LIN {X 0,Y 270.263,Z 149.626,A -85,B 0,C 180,E1 -17972.145,E2 -17972.145} C_VEL
LIN {X 0,Y 270.276,Z 149.627,A -85,B 0,C 180,E1 -17975.519,E2 -17975.519} C_VEL
LIN {X 0,Y 270.3,Z 149.622,A -85,B 0,C 180,E1 -17980.244,E2 -17980.244} C_VEL
LIN {X 0,Y 270.402,Z 149.614,A -85,B 0,C 180,E1 -17984.935,E2 -17984.935} C_VEL
LIN {X 0,Y 270.441,Z 149.602,A -85,B 0,C 180,E1 -17989.519,E2 -17989.519} C_VEL
LIN {X 0,Y 270.61,Z 149.58,A -85,B 0,C 180,E1 -17992.539,E2 -17992.539} C_VEL
LIN {X 0,Y 270.425,Z 149.61,A -85,B 0,C 180,E1 -17995.574,E2 -17995.574} C_VEL
LIN {X 0,Y 269.881,Z 149.678,A -85,B 0,C 180,E1 -17996.821,E2 -17996.821} C_VEL
LIN {X 0,Y 267.222,Z 150.002,A -85,B 0,C 180,E1 -17998.858,E2 -17998.858} C_VEL
LIN {X 0,Y 264.03,Z 150.39,A -85,B 0,C 180,E1 -18001.361,E2 -18001.361} C_VEL
LIN {X 0,Y 263.641,Z 150.441,A -85,B 0,C 180,E1 -18002.225,E2 -18002.225} C_VEL
LIN {X 0,Y 263.572,Z 150.462,A -85,B 0,C 180,E1 -18007.661,E2 -18007.661} C_VEL
LIN {X 0,Y 263.372,Z 150.472,A -85,B 0,C 180,E1 -18010.765,E2 -18010.765} C_VEL
LIN {X 0,Y 263.349,Z 150.494,A -85,B 0,C 180,E1 -18015.478,E2 -18015.478} C_VEL
LIN {X 0,Y 263.262,Z 150.491,A -85,B 0,C 180,E1 -18020.307,E2 -18020.307} C_VEL
LIN {X 0,Y 263.208,Z 150.508,A -85,B 0,C 180,E1 -18025.291,E2 -18025.291} C_VEL
LIN {X 0,Y 263.178,Z 150.505,A -85,B 0,C 180,E1 -18028.729,E2 -18028.729} C_VEL
LIN {X 0,Y 263.131,Z 150.521,A -85,B 0,C 180,E1 -18032.288,E2 -18032.288} C_VEL
LIN {X 0,Y 263.181,Z 150.514,A -85,B 0,C 180,E1 -18036.763,E2 -18036.763} C_VEL
LIN {X 0,Y 263.122,Z 150.503,A -85,B 0,C 180,E1 -18041.594,E2 -18041.594} C_VEL
LIN {X 0,Y 263.103,Z 150.515,A -85,B 0,C 180,E1 -18046.155,E2 -18046.155} C_VEL
LIN {X 0,Y 263.104,Z 150.514,A -85,B 0,C 180,E1 -18050.128,E2 -18050.128} C_VEL
LIN {X 0,Y 263.173,Z 150.515,A -85,B 0,C 180,E1 -18054.02,E2 -18054.02} C_VEL
LIN {X 0,Y 263.132,Z 150.511,A -85,B 0,C 180,E1 -18057.712,E2 -18057.712} C_VEL
LIN {X 0,Y 263.195,Z 150.632,A -85,B 0,C 180,E1 -18059.513,E2 -18059.513} C_VEL
LIN {X 0,Y 264.963,Z 158.96,A -85,B 0,C 180,E1 -18063.198,E2 -18063.198} C_VEL
LIN {X 0,Y 266.098,Z 165.732,A -85,B 0,C 180,E1 -18065.939,E2 -18065.939} C_VEL
LIN {X 0,Y 267.006,Z 169.677,A -85,B 0,C 180,E1 -18066.216,E2 -18066.216} C_VEL
LIN {X 0,Y 271.261,Z 194.933,A -85,B 0,C 180,E1 -18067.321,E2 -18067.321} C_VEL
LIN {X 0,Y 272.596,Z 205.287,A -85,B 0,C 180,E1 -18067.726,E2 -18067.726} C_VEL
LIN {X 0,Y 271.585,Z 243.518,A -85,B 0,C 180,E1 -18068.76,E2 -18068.76} C_VEL
LIN {X 0,Y 270.816,Z 255.136,A -85,B 0,C 180,E1 -18069.326,E2 -18069.326} C_VEL
LIN {X 0,Y 269.739,Z 266.296,A -85,B 0,C 180,E1 -18070.202,E2 -18070.202} C_VEL
LIN {X 0,Y 268.738,Z 274.976,A -85,B 0,C 180,E1 -18071.118,E2 -18071.118} C_VEL
LIN {X 0,Y 267.584,Z 283.269,A -85,B 0,C 180,E1 -18072.223,E2 -18072.223} C_VEL
LIN {X 0,Y 266.283,Z 291.12,A -85,B 0,C 180,E1 -18073.518,E2 -18073.518} C_VEL
LIN {X 0,Y 265.051,Z 298.464,A -85,B 0,C 180,E1 -18075.018,E2 -18075.018} C_VEL
LIN {X 0,Y 263.795,Z 305.915,A -85,B 0,C 180,E1 -18076.912,E2 -18076.912} C_VEL
LIN {X 0,Y 262.756,Z 311.756,A -85,B 0,C 180,E1 -18078.819,E2 -18078.819} C_VEL
LIN {X 0,Y 262.033,Z 316.362,A -85,B 0,C 180,E1 -18080.74,E2 -18080.74} C_VEL
LIN {X 0,Y 261.591,Z 319.357,A -85,B 0,C 180,E1 -18082.28,E2 -18082.28} C_VEL
LIN {X 0,Y 261.188,Z 322.632,A -85,B 0,C 180,E1 -18084.616,E2 -18084.616} C_VEL
LIN {X 0,Y 261.069,Z 324.672,A -85,B 0,C 180,E1 -18086.914,E2 -18086.914} C_VEL
LIN {X 0,Y 261.046,Z 325.447,A -85,B 0,C 180,E1 -18088.458,E2 -18088.458} C_VEL
LIN {X 0,Y 261.082,Z 325.74,A -85,B 0,C 180,E1 -18090,E2 -18090} C_VEL
LIN {X 0,Y 261.046,Z 325.44,A -85,B 0,C 180,E1 -18091.543,E2 -18091.543} C_VEL
LIN {X 0,Y 261.07,Z 324.65,A -85,B 0,C 180,E1 -18093.087,E2 -18093.087} C_VEL
LIN {X 0,Y 261.196,Z 322.574,A -85,B 0,C 180,E1 -18095.404,E2 -18095.404} C_VEL
LIN {X 0,Y 261.578,Z 319.298,A -85,B 0,C 180,E1 -18097.721,E2 -18097.721} C_VEL
LIN {X 0,Y 262.263,Z 314.543,A -85,B 0,C 180,E1 -18100.032,E2 -18100.032} C_VEL
LIN {X 0,Y 263.137,Z 309.397,A -85,B 0,C 180,E1 -18101.946,E2 -18101.946} C_VEL
LIN {X 0,Y 263.997,Z 304.366,A -85,B 0,C 180,E1 -18103.47,E2 -18103.47} C_VEL
LIN {X 0,Y 265.045,Z 298.308,A -85,B 0,C 180,E1 -18104.983,E2 -18104.983} C_VEL
LIN {X 0,Y 266.307,Z 290.937,A -85,B 0,C 180,E1 -18106.481,E2 -18106.481} C_VEL
LIN {X 0,Y 267.569,Z 283.043,A -85,B 0,C 180,E1 -18107.779,E2 -18107.779} C_VEL
LIN {X 0,Y 268.707,Z 274.696,A -85,B 0,C 180,E1 -18108.885,E2 -18108.885} C_VEL
LIN {X 0,Y 269.913,Z 264.253,A -85,B 0,C 180,E1 -18109.961,E2 -18109.961} C_VEL
LIN {X 0,Y 270.932,Z 252.949,A -85,B 0,C 180,E1 -18110.762,E2 -18110.762} C_VEL
LIN {X 0,Y 271.601,Z 243.673,A -85,B 0,C 180,E1 -18111.197,E2 -18111.197} C_VEL
LIN {X 0,Y 272.294,Z 214.479,A -85,B 0,C 180,E1 -18112.007,E2 -18112.007} C_VEL
LIN {X 0,Y 272.336,Z 202.812,A -85,B 0,C 180,E1 -18112.328,E2 -18112.328} C_VEL
LIN {X 0,Y 268.78,Z 179.455,A -85,B 0,C 180,E1 -18113.301,E2 -18113.301} C_VEL
LIN {X 0,Y 266.173,Z 166.332,A -85,B 0,C 180,E1 -18113.944,E2 -18113.944} C_VEL
LIN {X 0,Y 266.028,Z 165.241,A -85,B 0,C 180,E1 -18114.172,E2 -18114.172} C_VEL
LIN {X 0,Y 264.547,Z 156.793,A -85,B 0,C 180,E1 -18117.688,E2 -18117.688} C_VEL
LIN {X 0,Y 263.205,Z 150.537,A -85,B 0,C 180,E1 -18120.523,E2 -18120.523} C_VEL
LIN {X 0,Y 263.152,Z 150.51,A -85,B 0,C 180,E1 -18124.115,E2 -18124.115} C_VEL
LIN {X 0,Y 263.162,Z 150.499,A -85,B 0,C 180,E1 -18127.897,E2 -18127.897} C_VEL
LIN {X 0,Y 263.124,Z 150.524,A -85,B 0,C 180,E1 -18131.894,E2 -18131.894} C_VEL
LIN {X 0,Y 263.105,Z 150.489,A -85,B 0,C 180,E1 -18136.155,E2 -18136.155} C_VEL
LIN {X 0,Y 263.106,Z 150.522,A -85,B 0,C 180,E1 -18140.128,E2 -18140.128} C_VEL
LIN {X 0,Y 263.164,Z 150.51,A -85,B 0,C 180,E1 -18144.018,E2 -18144.018} C_VEL
LIN {X 0,Y 263.134,Z 150.521,A -85,B 0,C 180,E1 -18147.712,E2 -18147.712} C_VEL
LIN {X 0,Y 263.203,Z 150.498,A -85,B 0,C 180,E1 -18151.783,E2 -18151.783} C_VEL
LIN {X 0,Y 263.228,Z 150.51,A -85,B 0,C 180,E1 -18155.2,E2 -18155.2} C_VEL
LIN {X 0,Y 263.265,Z 150.49,A -85,B 0,C 180,E1 -18159.694,E2 -18159.694} C_VEL
LIN {X 0,Y 263.353,Z 150.494,A -85,B 0,C 180,E1 -18164.522,E2 -18164.522} C_VEL
LIN {X 0,Y 263.357,Z 150.474,A -85,B 0,C 180,E1 -18169.234,E2 -18169.234} C_VEL
LIN {X 0,Y 263.56,Z 150.463,A -85,B 0,C 180,E1 -18172.338,E2 -18172.338} C_VEL
LIN {X 0,Y 263.752,Z 150.426,A -85,B 0,C 180,E1 -18178.473,E2 -18178.473} C_VEL
LIN {X 0,Y 263.753,Z 150.435,A -85,B 0,C 180,E1 -18181.527,E2 -18181.527} C_VEL
LIN {X 0,Y 263.575,Z 150.453,A -85,B 0,C 180,E1 -18187.662,E2 -18187.662} C_VEL
LIN {X 0,Y 263.377,Z 150.481,A -85,B 0,C 180,E1 -18190.766,E2 -18190.766} C_VEL
LIN {X 0,Y 263.353,Z 150.49,A -85,B 0,C 180,E1 -18195.478,E2 -18195.478} C_VEL
LIN {X 0,Y 263.266,Z 150.497,A -85,B 0,C 180,E1 -18200.307,E2 -18200.307} C_VEL
LIN {X 0,Y 263.21,Z 150.501,A -85,B 0,C 180,E1 -18205.291,E2 -18205.291} C_VEL
LIN {X 0,Y 263.181,Z 150.51,A -85,B 0,C 180,E1 -18208.73,E2 -18208.73} C_VEL
LIN {X 0,Y 263.135,Z 150.518,A -85,B 0,C 180,E1 -18212.288,E2 -18212.288} C_VEL
LIN {X 0,Y 263.185,Z 150.516,A -85,B 0,C 180,E1 -18216.763,E2 -18216.763} C_VEL
LIN {X 0,Y 263.126,Z 150.519,A -85,B 0,C 180,E1 -18221.593,E2 -18221.593} C_VEL
LIN {X 0,Y 263.124,Z 150.522,A -85,B 0,C 180,E1 -18223.984,E2 -18223.984} C_VEL
LIN {X 0,Y 263.126,Z 150.497,A -85,B 0,C 180,E1 -18228.406,E2 -18228.406} C_VEL
LIN {X 0,Y 263.167,Z 150.517,A -85,B 0,C 180,E1 -18232.104,E2 -18232.104} C_VEL
LIN {X 0,Y 263.169,Z 150.498,A -85,B 0,C 180,E1 -18235.888,E2 -18235.888} C_VEL
LIN {X 0,Y 263.153,Z 150.511,A -85,B 0,C 180,E1 -18239.507,E2 -18239.507} C_VEL
LIN {X 0,Y 263.297,Z 150.677,A -85,B 0,C 180,E1 -18243.014,E2 -18243.014} C_VEL
LIN {X 0,Y 264.578,Z 157.239,A -85,B 0,C 180,E1 -18245.894,E2 -18245.894} C_VEL
LIN {X 0,Y 266.07,Z 161.339,A -85,B 0,C 180,E1 -18246.226,E2 -18246.226} C_VEL
LIN {X 0,Y 269.712,Z 171.853,A -85,B 0,C 180,E1 -18246.868,E2 -18246.868} C_VEL
LIN {X 0,Y 272.813,Z 188.856,A -85,B 0,C 180,E1 -18247.623,E2 -18247.623} C_VEL
LIN {X 0,Y 271.762,Z 233.501,A -85,B 0,C 180,E1 -18248.823,E2 -18248.823} C_VEL
LIN {X 0,Y 271.245,Z 243.265,A -85,B 0,C 180,E1 -18249.278,E2 -18249.278} C_VEL
LIN {X 0,Y 270.43,Z 254.338,A -85,B 0,C 180,E1 -18250.056,E2 -18250.056} C_VEL
LIN {X 0,Y 269.192,Z 265.146,A -85,B 0,C 180,E1 -18251.15,E2 -18251.15} C_VEL
LIN {X 0,Y 268.087,Z 273.533,A -85,B 0,C 180,E1 -18252.256,E2 -18252.256} C_VEL
LIN {X 0,Y 266.877,Z 281.453,A -85,B 0,C 180,E1 -18253.555,E2 -18253.555} C_VEL
LIN {X 0,Y 265.981,Z 287.139,A -85,B 0,C 180,E1 -18254.679,E2 -18254.679} C_VEL
LIN {X 0,Y 264.849,Z 293.489,A -85,B 0,C 180,E1 -18256.183,E2 -18256.183} C_VEL
LIN {X 0,Y 263.923,Z 298.766,A -85,B 0,C 180,E1 -18257.7,E2 -18257.7} C_VEL
LIN {X 0,Y 263.077,Z 303.172,A -85,B 0,C 180,E1 -18259.222,E2 -18259.222} C_VEL
LIN {X 0,Y 262.253,Z 308.35,A -85,B 0,C 180,E1 -18261.524,E2 -18261.524} C_VEL
LIN {X 0,Y 261.681,Z 311.772,A -85,B 0,C 180,E1 -18263.574,E2 -18263.574} C_VEL
LIN {X 0,Y 261.381,Z 313.917,A -85,B 0,C 180,E1 -18265.373,E2 -18265.373} C_VEL
LIN {X 0,Y 261.213,Z 315.186,A -85,B 0,C 180,E1 -18266.915,E2 -18266.915} C_VEL
LIN {X 0,Y 261.099,Z 315.987,A -85,B 0,C 180,E1 -18268.457,E2 -18268.457} C_VEL
LIN {X 0,Y 261.088,Z 316.292,A -85,B 0,C 180,E1 -18270,E2 -18270} C_VEL
LIN {X 0,Y 261.099,Z 316.013,A -85,B 0,C 180,E1 -18271.542,E2 -18271.542} C_VEL
LIN {X 0,Y 261.211,Z 315.265,A -85,B 0,C 180,E1 -18273.084,E2 -18273.084} C_VEL
LIN {X 0,Y 261.371,Z 314.049,A -85,B 0,C 180,E1 -18274.627,E2 -18274.627} C_VEL
LIN {X 0,Y 261.755,Z 311.196,A -85,B 0,C 180,E1 -18276.938,E2 -18276.938} C_VEL
LIN {X 0,Y 262.2,Z 308.596,A -85,B 0,C 180,E1 -18278.477,E2 -18278.477} C_VEL
LIN {X 0,Y 263.061,Z 303.484,A -85,B 0,C 180,E1 -18280.778,E2 -18280.778} C_VEL
LIN {X 0,Y 264.072,Z 297.981,A -85,B 0,C 180,E1 -18282.683,E2 -18282.683} C_VEL
LIN {X 0,Y 265.345,Z 291.064,A -85,B 0,C 180,E1 -18284.573,E2 -18284.573} C_VEL
LIN {X 0,Y 266.64,Z 283.123,A -85,B 0,C 180,E1 -18286.263,E2 -18286.263} C_VEL
LIN {X 0,Y 267.825,Z 275.549,A -85,B 0,C 180,E1 -18287.564,E2 -18287.564} C_VEL
LIN {X 0,Y 268.995,Z 267.606,A -85,B 0,C 180,E1 -18288.666,E2 -18288.666} C_VEL
LIN {X 0,Y 269.999,Z 259.4,A -85,B 0,C 180,E1 -18289.58,E2 -18289.58} C_VEL
LIN {X 0,Y 270.786,Z 251.226,A -85,B 0,C 180,E1 -18290.3,E2 -18290.3} C_VEL
LIN {X 0,Y 271.431,Z 242.496,A -85,B 0,C 180,E1 -18290.88,E2 -18290.88} C_VEL
LIN {X 0,Y 271.86,Z 234.107,A -85,B 0,C 180,E1 -18291.272,E2 -18291.272} C_VEL
LIN {X 0,Y 272.318,Z 212.774,A -85,B 0,C 180,E1 -18291.88,E2 -18291.88} C_VEL
LIN {X 0,Y 272.859,Z 188.975,A -85,B 0,C 180,E1 -18292.497,E2 -18292.497} C_VEL
LIN {X 0,Y 269.51,Z 171.11,A -85,B 0,C 180,E1 -18293.301,E2 -18293.301} C_VEL
LIN {X 0,Y 265.613,Z 160.117,A -85,B 0,C 180,E1 -18293.984,E2 -18293.984} C_VEL
LIN {X 0,Y 264.555,Z 157.188,A -85,B 0,C 180,E1 -18294.249,E2 -18294.249} C_VEL
LIN {X 0,Y 263.312,Z 150.747,A -85,B 0,C 180,E1 -18297.078,E2 -18297.078} C_VEL
LIN {X 0,Y 263.18,Z 150.515,A -85,B 0,C 180,E1 -18298.729,E2 -18298.729} C_VEL
LIN {X 0,Y 263.134,Z 150.522,A -85,B 0,C 180,E1 -18302.288,E2 -18302.288} C_VEL
LIN {X 0,Y 263.187,Z 150.497,A -85,B 0,C 180,E1 -18305.977,E2 -18305.977} C_VEL
LIN {X 0,Y 263.115,Z 150.517,A -85,B 0,C 180,E1 -18309.87,E2 -18309.87} C_VEL
LIN {X 0,Y 263.103,Z 150.504,A -85,B 0,C 180,E1 -18313.988,E2 -18313.988} C_VEL
LIN {X 0,Y 263.123,Z 150.521,A -85,B 0,C 180,E1 -18318.106,E2 -18318.106} C_VEL
LIN {X 0,Y 263.158,Z 150.516,A -85,B 0,C 180,E1 -18322.103,E2 -18322.103} C_VEL
LIN {X 0,Y 263.15,Z 150.507,A -85,B 0,C 180,E1 -18325.885,E2 -18325.885} C_VEL
LIN {X 0,Y 263.15,Z 150.519,A -85,B 0,C 180,E1 -18329.507,E2 -18329.507} C_VEL
LIN {X 0,Y 263.191,Z 150.502,A -85,B 0,C 180,E1 -18333.002,E2 -18333.002} C_VEL
LIN {X 0,Y 263.183,Z 150.511,A -85,B 0,C 180,E1 -18336.387,E2 -18336.387} C_VEL
LIN {X 0,Y 263.263,Z 150.498,A -85,B 0,C 180,E1 -18339.693,E2 -18339.693} C_VEL
LIN {X 0,Y 263.35,Z 150.49,A -85,B 0,C 180,E1 -18344.522,E2 -18344.522} C_VEL
LIN {X 0,Y 263.373,Z 150.481,A -85,B 0,C 180,E1 -18349.234,E2 -18349.234} C_VEL
LIN {X 0,Y 263.571,Z 150.453,A -85,B 0,C 180,E1 -18352.338,E2 -18352.338} C_VEL
LIN {X 0,Y 263.751,Z 150.436,A -85,B 0,C 180,E1 -18358.473,E2 -18358.473} C_VEL
LIN {X 0,Y 263.75,Z 150.426,A -85,B 0,C 180,E1 -18361.527,E2 -18361.527} C_VEL
LIN {X 0,Y 263.641,Z 150.441,A -85,B 0,C 180,E1 -18362.225,E2 -18362.225} C_VEL
LIN {X 0,Y 262.865,Z 150.549,A -85,B 0,C 180,E1 -18363.499,E2 -18363.499} C_VEL
LIN {X 0,Y 259.97,Z 150.915,A -85,B 0,C 180,E1 -18365.576,E2 -18365.576} C_VEL
LIN {X 0,Y 257.579,Z 151.211,A -85,B 0,C 180,E1 -18367.264,E2 -18367.264} C_VEL
LIN {X 0,Y 256.559,Z 151.33,A -85,B 0,C 180,E1 -18368.574,E2 -18368.574} C_VEL
LIN {X 0,Y 256.476,Z 151.335,A -85,B 0,C 180,E1 -18369.017,E2 -18369.017} C_VEL
LIN {X 0,Y 256.294,Z 151.365,A -85,B 0,C 180,E1 -18372.672,E2 -18372.672} C_VEL
LIN {X 0,Y 256.281,Z 151.371,A -85,B 0,C 180,E1 -18376.302,E2 -18376.302} C_VEL
LIN {X 0,Y 256.156,Z 151.38,A -85,B 0,C 180,E1 -18381.12,E2 -18381.12} C_VEL
LIN {X 0,Y 256.187,Z 151.383,A -85,B 0,C 180,E1 -18385.139,E2 -18385.139} C_VEL
LIN {X 0,Y 256.112,Z 151.392,A -85,B 0,C 180,E1 -18389.6,E2 -18389.6} C_VEL
LIN {X 0,Y 256.066,Z 151.395,A -85,B 0,C 180,E1 -18393.293,E2 -18393.293} C_VEL
LIN {X 0,Y 256.113,Z 151.395,A -85,B 0,C 180,E1 -18397.271,E2 -18397.271} C_VEL
LIN {X 0,Y 256.052,Z 151.387,A -85,B 0,C 180,E1 -18401.204,E2 -18401.204} C_VEL
LIN {X 0,Y 256.039,Z 151.391,A -85,B 0,C 180,E1 -18405.534,E2 -18405.534} C_VEL
LIN {X 0,Y 256.053,Z 151.4,A -85,B 0,C 180,E1 -18408.797,E2 -18408.797} C_VEL
LIN {X 0,Y 256.134,Z 151.379,A -85,B 0,C 180,E1 -18412.869,E2 -18412.869} C_VEL
LIN {X 0,Y 256.067,Z 151.388,A -85,B 0,C 180,E1 -18416.708,E2 -18416.708} C_VEL
LIN {X 0,Y 256.126,Z 151.528,A -85,B 0,C 180,E1 -18419.037,E2 -18419.037} C_VEL
LIN {X 0,Y 257.709,Z 158.819,A -85,B 0,C 180,E1 -18422.38,E2 -18422.38} C_VEL
LIN {X 0,Y 258.959,Z 165.635,A -85,B 0,C 180,E1 -18425.239,E2 -18425.239} C_VEL
LIN {X 0,Y 260.509,Z 170.647,A -85,B 0,C 180,E1 -18425.616,E2 -18425.616} C_VEL
LIN {X 0,Y 265.165,Z 198.563,A -85,B 0,C 180,E1 -18426.877,E2 -18426.877} C_VEL
LIN {X 0,Y 266.018,Z 205.812,A -85,B 0,C 180,E1 -18427.163,E2 -18427.163} C_VEL
LIN {X 0,Y 265.042,Z 242.239,A -85,B 0,C 180,E1 -18428.163,E2 -18428.163} C_VEL
LIN {X 0,Y 264.452,Z 251.768,A -85,B 0,C 180,E1 -18428.602,E2 -18428.602} C_VEL
LIN {X 0,Y 263.459,Z 262.934,A -85,B 0,C 180,E1 -18429.38,E2 -18429.38} C_VEL
LIN {X 0,Y 262.208,Z 273.349,A -85,B 0,C 180,E1 -18430.426,E2 -18430.426} C_VEL
LIN {X 0,Y 261.025,Z 281.914,A -85,B 0,C 180,E1 -18431.557,E2 -18431.557} C_VEL
LIN {X 0,Y 259.635,Z 289.972,A -85,B 0,C 180,E1 -18432.881,E2 -18432.881} C_VEL
LIN {X 0,Y 258.496,Z 296.631,A -85,B 0,C 180,E1 -18434.224,E2 -18434.224} C_VEL
LIN {X 0,Y 257.33,Z 302.953,A -85,B 0,C 180,E1 -18435.771,E2 -18435.771} C_VEL
LIN {X 0,Y 256.389,Z 308.207,A -85,B 0,C 180,E1 -18437.333,E2 -18437.333} C_VEL
LIN {X 0,Y 255.609,Z 312.588,A -85,B 0,C 180,E1 -18438.904,E2 -18438.904} C_VEL
LIN {X 0,Y 254.777,Z 317.758,A -85,B 0,C 180,E1 -18441.274,E2 -18441.274} C_VEL
LIN {X 0,Y 254.207,Z 321.552,A -85,B 0,C 180,E1 -18443.651,E2 -18443.651} C_VEL
LIN {X 0,Y 254.061,Z 323.296,A -85,B 0,C 180,E1 -18445.24,E2 -18445.24} C_VEL
LIN {X 0,Y 253.972,Z 324.544,A -85,B 0,C 180,E1 -18446.828,E2 -18446.828} C_VEL
LIN {X 0,Y 253.957,Z 325.319,A -85,B 0,C 180,E1 -18448.415,E2 -18448.415} C_VEL
LIN {X 0,Y 253.989,Z 325.612,A -85,B 0,C 180,E1 -18450,E2 -18450} C_VEL
LIN {X 0,Y 253.957,Z 325.311,A -85,B 0,C 180,E1 -18451.586,E2 -18451.586} C_VEL
LIN {X 0,Y 253.972,Z 324.521,A -85,B 0,C 180,E1 -18453.173,E2 -18453.173} C_VEL
LIN {X 0,Y 254.085,Z 322.726,A -85,B 0,C 180,E1 -18455.279,E2 -18455.279} C_VEL
LIN {X 0,Y 254.544,Z 319.168,A -85,B 0,C 180,E1 -18457.935,E2 -18457.935} C_VEL
LIN {X 0,Y 255.256,Z 314.413,A -85,B 0,C 180,E1 -18460.31,E2 -18460.31} C_VEL
LIN {X 0,Y 256.171,Z 309.266,A -85,B 0,C 180,E1 -18462.276,E2 -18462.276} C_VEL
LIN {X 0,Y 257.076,Z 304.235,A -85,B 0,C 180,E1 -18463.84,E2 -18463.84} C_VEL
LIN {X 0,Y 258.169,Z 298.177,A -85,B 0,C 180,E1 -18465.392,E2 -18465.392} C_VEL
LIN {X 0,Y 259.502,Z 290.806,A -85,B 0,C 180,E1 -18466.926,E2 -18466.926} C_VEL
LIN {X 0,Y 260.825,Z 282.911,A -85,B 0,C 180,E1 -18468.255,E2 -18468.255} C_VEL
LIN {X 0,Y 261.998,Z 274.563,A -85,B 0,C 180,E1 -18469.388,E2 -18469.388} C_VEL
LIN {X 0,Y 263.233,Z 264.33,A -85,B 0,C 180,E1 -18470.469,E2 -18470.469} C_VEL
LIN {X 0,Y 264.313,Z 252.944,A -85,B 0,C 180,E1 -18471.299,E2 -18471.299} C_VEL
LIN {X 0,Y 265,Z 243.247,A -85,B 0,C 180,E1 -18471.762,E2 -18471.762} C_VEL
LIN {X 0,Y 265.875,Z 204.461,A -85,B 0,C 180,E1 -18472.85,E2 -18472.85} C_VEL
LIN {X 0,Y 262.258,Z 180.54,A -85,B 0,C 180,E1 -18473.88,E2 -18473.88} C_VEL
LIN {X 0,Y 259.863,Z 168.483,A -85,B 0,C 180,E1 -18474.47,E2 -18474.47} C_VEL
LIN {X 0,Y 258.933,Z 165.659,A -85,B 0,C 180,E1 -18474.718,E2 -18474.718} C_VEL
LIN {X 0,Y 257.699,Z 158.712,A -85,B 0,C 180,E1 -18477.622,E2 -18477.622} C_VEL
LIN {X 0,Y 256.14,Z 151.436,A -85,B 0,C 180,E1 -18480.991,E2 -18480.991} C_VEL
LIN {X 0,Y 256.089,Z 151.398,A -85,B 0,C 180,E1 -18485.192,E2 -18485.192} C_VEL
LIN {X 0,Y 256.121,Z 151.379,A -85,B 0,C 180,E1 -18487.273,E2 -18487.273} C_VEL
LIN {X 0,Y 256.055,Z 151.4,A -85,B 0,C 180,E1 -18491.204,E2 -18491.204} C_VEL
LIN {X 0,Y 256.041,Z 151.371,A -85,B 0,C 180,E1 -18495.534,E2 -18495.534} C_VEL
LIN {X 0,Y 256.055,Z 151.388,A -85,B 0,C 180,E1 -18498.797,E2 -18498.797} C_VEL
LIN {X 0,Y 256.132,Z 151.392,A -85,B 0,C 180,E1 -18502.868,E2 -18502.868} C_VEL
LIN {X 0,Y 256.069,Z 151.395,A -85,B 0,C 180,E1 -18506.708,E2 -18506.708} C_VEL
LIN {X 0,Y 256.115,Z 151.391,A -85,B 0,C 180,E1 -18510.401,E2 -18510.401} C_VEL
LIN {X 0,Y 256.19,Z 151.383,A -85,B 0,C 180,E1 -18514.861,E2 -18514.861} C_VEL
LIN {X 0,Y 256.168,Z 151.376,A -85,B 0,C 180,E1 -18519.105,E2 -18519.105} C_VEL
LIN {X 0,Y 256.302,Z 151.37,A -85,B 0,C 180,E1 -18524.085,E2 -18524.085} C_VEL
LIN {X 0,Y 256.299,Z 151.353,A -85,B 0,C 180,E1 -18528.934,E2 -18528.934} C_VEL
LIN {X 0,Y 256.517,Z 151.338,A -85,B 0,C 180,E1 -18532.127,E2 -18532.127} C_VEL
LIN {X 0,Y 256.499,Z 151.339,A -85,B 0,C 180,E1 -18536.859,E2 -18536.859} C_VEL
LIN {X 0,Y 256.76,Z 151.296,A -85,B 0,C 180,E1 -18540,E2 -18540} C_VEL
LIN {X 0,Y 256.5,Z 151.344,A -85,B 0,C 180,E1 -18543.142,E2 -18543.142} C_VEL
LIN {X 0,Y 256.542,Z 151.326,A -85,B 0,C 180,E1 -18547.873,E2 -18547.873} C_VEL
LIN {X 0,Y 256.313,Z 151.361,A -85,B 0,C 180,E1 -18551.066,E2 -18551.066} C_VEL
LIN {X 0,Y 256.302,Z 151.365,A -85,B 0,C 180,E1 -18555.915,E2 -18555.915} C_VEL
LIN {X 0,Y 256.169,Z 151.383,A -85,B 0,C 180,E1 -18560.895,E2 -18560.895} C_VEL
LIN {X 0,Y 256.19,Z 151.376,A -85,B 0,C 180,E1 -18565.138,E2 -18565.138} C_VEL
LIN {X 0,Y 256.116,Z 151.394,A -85,B 0,C 180,E1 -18569.6,E2 -18569.6} C_VEL
LIN {X 0,Y 256.07,Z 151.388,A -85,B 0,C 180,E1 -18573.293,E2 -18573.293} C_VEL
LIN {X 0,Y 256.117,Z 151.394,A -85,B 0,C 180,E1 -18577.271,E2 -18577.271} C_VEL
LIN {X 0,Y 256.056,Z 151.4,A -85,B 0,C 180,E1 -18581.203,E2 -18581.203} C_VEL
LIN {X 0,Y 256.046,Z 151.391,A -85,B 0,C 180,E1 -18585.533,E2 -18585.533} C_VEL
LIN {X 0,Y 256.058,Z 151.379,A -85,B 0,C 180,E1 -18588.797,E2 -18588.797} C_VEL
LIN {X 0,Y 256.146,Z 151.387,A -85,B 0,C 180,E1 -18592.87,E2 -18592.87} C_VEL
LIN {X 0,Y 256.078,Z 151.39,A -85,B 0,C 180,E1 -18596.708,E2 -18596.708} C_VEL
LIN {X 0,Y 256.141,Z 151.392,A -85,B 0,C 180,E1 -18601.404,E2 -18601.404} C_VEL
LIN {X 0,Y 256.265,Z 151.551,A -85,B 0,C 180,E1 -18602.543,E2 -18602.543} C_VEL
LIN {X 0,Y 257.41,Z 157.377,A -85,B 0,C 180,E1 -18605.177,E2 -18605.177} C_VEL
LIN {X 0,Y 258.898,Z 161.415,A -85,B 0,C 180,E1 -18605.522,E2 -18605.522} C_VEL
LIN {X 0,Y 263.102,Z 172.815,A -85,B 0,C 180,E1 -18606.275,E2 -18606.275} C_VEL
LIN {X 0,Y 266.181,Z 189.334,A -85,B 0,C 180,E1 -18607.043,E2 -18607.043} C_VEL
LIN {X 0,Y 265.392,Z 227.395,A -85,B 0,C 180,E1 -18608.064,E2 -18608.064} C_VEL
LIN {X 0,Y 264.843,Z 240.179,A -85,B 0,C 180,E1 -18608.555,E2 -18608.555} C_VEL
LIN {X 0,Y 264.174,Z 249.7,A -85,B 0,C 180,E1 -18609.159,E2 -18609.159} C_VEL
LIN {X 0,Y 263.367,Z 258.335,A -85,B 0,C 180,E1 -18609.905,E2 -18609.905} C_VEL
LIN {X 0,Y 262.298,Z 266.777,A -85,B 0,C 180,E1 -18610.839,E2 -18610.839} C_VEL
LIN {X 0,Y 261.148,Z 274.894,A -85,B 0,C 180,E1 -18611.971,E2 -18611.971} C_VEL
LIN {X 0,Y 259.941,Z 282.604,A -85,B 0,C 180,E1 -18613.305,E2 -18613.305} C_VEL
LIN {X 0,Y 258.556,Z 290.666,A -85,B 0,C 180,E1 -18615.035,E2 -18615.035} C_VEL
LIN {X 0,Y 257.193,Z 297.727,A -85,B 0,C 180,E1 -18616.971,E2 -18616.971} C_VEL
LIN {X 0,Y 256.09,Z 303.303,A -85,B 0,C 180,E1 -18618.924,E2 -18618.924} C_VEL
LIN {X 0,Y 255.227,Z 308.48,A -85,B 0,C 180,E1 -18621.289,E2 -18621.289} C_VEL
LIN {X 0,Y 254.605,Z 312.168,A -85,B 0,C 180,E1 -18623.58,E2 -18623.58} C_VEL
LIN {X 0,Y 254.304,Z 314.046,A -85,B 0,C 180,E1 -18625.244,E2 -18625.244} C_VEL
LIN {X 0,Y 254.135,Z 315.315,A -85,B 0,C 180,E1 -18626.829,E2 -18626.829} C_VEL
LIN {X 0,Y 254.011,Z 316.116,A -85,B 0,C 180,E1 -18628.414,E2 -18628.414} C_VEL
LIN {X 0,Y 254.018,Z 316.42,A -85,B 0,C 180,E1 -18630,E2 -18630} C_VEL
LIN {X 0,Y 254.011,Z 316.141,A -85,B 0,C 180,E1 -18631.585,E2 -18631.585} C_VEL
LIN {X 0,Y 254.132,Z 315.393,A -85,B 0,C 180,E1 -18633.17,E2 -18633.17} C_VEL
LIN {X 0,Y 254.291,Z 314.176,A -85,B 0,C 180,E1 -18634.756,E2 -18634.756} C_VEL
LIN {X 0,Y 254.53,Z 312.47,A -85,B 0,C 180,E1 -18636.341,E2 -18636.341} C_VEL
LIN {X 0,Y 255.189,Z 308.723,A -85,B 0,C 180,E1 -18638.712,E2 -18638.712} C_VEL
LIN {X 0,Y 256.078,Z 303.611,A -85,B 0,C 180,E1 -18641.076,E2 -18641.076} C_VEL
LIN {X 0,Y 257.139,Z 298.107,A -85,B 0,C 180,E1 -18643.031,E2 -18643.031} C_VEL
LIN {X 0,Y 258.496,Z 291.19,A -85,B 0,C 180,E1 -18644.968,E2 -18644.968} C_VEL
LIN {X 0,Y 259.833,Z 283.248,A -85,B 0,C 180,E1 -18646.701,E2 -18646.701} C_VEL
LIN {X 0,Y 261.087,Z 275.673,A -85,B 0,C 180,E1 -18648.032,E2 -18648.032} C_VEL
LIN {X 0,Y 262.296,Z 267.729,A -85,B 0,C 180,E1 -18649.161,E2 -18649.161} C_VEL
LIN {X 0,Y 263.343,Z 259.522,A -85,B 0,C 180,E1 -18650.096,E2 -18650.096} C_VEL
LIN {X 0,Y 264.235,Z 250.538,A -85,B 0,C 180,E1 -18650.894,E2 -18650.894} C_VEL
LIN {X 0,Y 264.914,Z 241.079,A -85,B 0,C 180,E1 -18651.513,E2 -18651.513} C_VEL
LIN {X 0,Y 265.318,Z 230.589,A -85,B 0,C 180,E1 -18651.966,E2 -18651.966} C_VEL
LIN {X 0,Y 266.315,Z 189.944,A -85,B 0,C 180,E1 -18653.056,E2 -18653.056} C_VEL
LIN {X 0,Y 263.257,Z 173.419,A -85,B 0,C 180,E1 -18653.823,E2 -18653.823} C_VEL
LIN {X 0,Y 259.585,Z 163.09,A -85,B 0,C 180,E1 -18654.491,E2 -18654.491} C_VEL
LIN {X 0,Y 257.467,Z 157.603,A -85,B 0,C 180,E1 -18654.916,E2 -18654.916} C_VEL
LIN {X 0,Y 257.227,Z 156.464,A -85,B 0,C 180,E1 -18655.272,E2 -18655.272} C_VEL
LIN {X 0,Y 256.213,Z 151.476,A -85,B 0,C 180,E1 -18657.684,E2 -18657.684} C_VEL
LIN {X 0,Y 256.084,Z 151.398,A -85,B 0,C 180,E1 -18661.704,E2 -18661.704} C_VEL
LIN {X 0,Y 256.12,Z 151.372,A -85,B 0,C 180,E1 -18665.186,E2 -18665.186} C_VEL
LIN {X 0,Y 256.088,Z 151.397,A -85,B 0,C 180,E1 -18669.138,E2 -18669.138} C_VEL
LIN {X 0,Y 256.048,Z 151.373,A -85,B 0,C 180,E1 -18673.329,E2 -18673.329} C_VEL
LIN {X 0,Y 256.071,Z 151.401,A -85,B 0,C 180,E1 -18677.818,E2 -18677.818} C_VEL
LIN {X 0,Y 256.07,Z 151.392,A -85,B 0,C 180,E1 -18680.858,E2 -18680.858} C_VEL
LIN {X 0,Y 256.13,Z 151.393,A -85,B 0,C 180,E1 -18682.867,E2 -18682.867} C_VEL
LIN {X 0,Y 256.067,Z 151.388,A -85,B 0,C 180,E1 -18686.707,E2 -18686.707} C_VEL
LIN {X 0,Y 256.113,Z 151.394,A -85,B 0,C 180,E1 -18690.4,E2 -18690.4} C_VEL
LIN {X 0,Y 256.187,Z 151.376,A -85,B 0,C 180,E1 -18694.861,E2 -18694.861} C_VEL
LIN {X 0,Y 256.166,Z 151.384,A -85,B 0,C 180,E1 -18699.105,E2 -18699.105} C_VEL
LIN {X 0,Y 256.299,Z 151.364,A -85,B 0,C 180,E1 -18704.085,E2 -18704.085} C_VEL
LIN {X 0,Y 256.309,Z 151.362,A -85,B 0,C 180,E1 -18708.934,E2 -18708.934} C_VEL
LIN {X 0,Y 256.539,Z 151.326,A -85,B 0,C 180,E1 -18712.127,E2 -18712.127} C_VEL
LIN {X 0,Y 256.713,Z 151.312,A -85,B 0,C 180,E1 -18718.431,E2 -18718.431} C_VEL
LIN {X 0,Y 256.713,Z 151.301,A -85,B 0,C 180,E1 -18721.569,E2 -18721.569} C_VEL
LIN {X 0,Y 256.539,Z 151.336,A -85,B 0,C 180,E1 -18727.873,E2 -18727.873} C_VEL
LIN {X 0,Y 256.476,Z 151.335,A -85,B 0,C 180,E1 -18729.017,E2 -18729.017} C_VEL
LIN {X 0,Y 255.772,Z 151.423,A -85,B 0,C 180,E1 -18730.326,E2 -18730.326} C_VEL
LIN {X 0,Y 252.797,Z 151.8,A -85,B 0,C 180,E1 -18732.455,E2 -18732.455} C_VEL
LIN {X 0,Y 250.303,Z 152.117,A -85,B 0,C 180,E1 -18734.189,E2 -18734.189} C_VEL
LIN {X 0,Y 249.275,Z 152.247,A -85,B 0,C 180,E1 -18735.537,E2 -18735.537} C_VEL
LIN {X 0,Y 249.213,Z 152.25,A -85,B 0,C 180,E1 -18735.994,E2 -18735.994} C_VEL
LIN {X 0,Y 249.109,Z 152.251,A -85,B 0,C 180,E1 -18739.788,E2 -18739.788} C_VEL
LIN {X 0,Y 249.15,Z 152.26,A -85,B 0,C 180,E1 -18745.031,E2 -18745.031} C_VEL
LIN {X 0,Y 249.082,Z 152.262,A -85,B 0,C 180,E1 -18748.994,E2 -18748.994} C_VEL
LIN {X 0,Y 249.029,Z 152.278,A -85,B 0,C 180,E1 -18752.426,E2 -18752.426} C_VEL
LIN {X 0,Y 249.046,Z 152.27,A -85,B 0,C 180,E1 -18756.342,E2 -18756.342} C_VEL
LIN {X 0,Y 249.004,Z 152.268,A -85,B 0,C 180,E1 -18760.478,E2 -18760.478} C_VEL
LIN {X 0,Y 248.983,Z 152.255,A -85,B 0,C 180,E1 -18764.883,E2 -18764.883} C_VEL
LIN {X 0,Y 249.008,Z 152.278,A -85,B 0,C 180,E1 -18767.362,E2 -18767.362} C_VEL
LIN {X 0,Y 249.026,Z 152.257,A -85,B 0,C 180,E1 -18771.62,E2 -18771.62} C_VEL
LIN {X 0,Y 249.044,Z 152.269,A -85,B 0,C 180,E1 -18775.64,E2 -18775.64} C_VEL
LIN {X 0,Y 249.07,Z 152.424,A -85,B 0,C 180,E1 -18778.533,E2 -18778.533} C_VEL
LIN {X 0,Y 250.685,Z 159.727,A -85,B 0,C 180,E1 -18781.993,E2 -18781.993} C_VEL
LIN {X 0,Y 251.78,Z 165.508,A -85,B 0,C 180,E1 -18784.485,E2 -18784.485} C_VEL
LIN {X 0,Y 253.816,Z 171.355,A -85,B 0,C 180,E1 -18784.955,E2 -18784.955} C_VEL
LIN {X 0,Y 256.597,Z 186.358,A -85,B 0,C 180,E1 -18785.695,E2 -18785.695} C_VEL
LIN {X 0,Y 259.485,Z 206.407,A -85,B 0,C 180,E1 -18786.575,E2 -18786.575} C_VEL
LIN {X 0,Y 258.484,Z 241.852,A -85,B 0,C 180,E1 -18787.568,E2 -18787.568} C_VEL
LIN {X 0,Y 257.882,Z 251.094,A -85,B 0,C 180,E1 -18787.994,E2 -18787.994} C_VEL
LIN {X 0,Y 257.073,Z 260.281,A -85,B 0,C 180,E1 -18788.623,E2 -18788.623} C_VEL
LIN {X 0,Y 255.96,Z 269.798,A -85,B 0,C 180,E1 -18789.508,E2 -18789.508} C_VEL
LIN {X 0,Y 254.481,Z 280.557,A -85,B 0,C 180,E1 -18790.856,E2 -18790.856} C_VEL
LIN {X 0,Y 253.078,Z 288.825,A -85,B 0,C 180,E1 -18792.214,E2 -18792.214} C_VEL
LIN {X 0,Y 251.666,Z 296.505,A -85,B 0,C 180,E1 -18793.784,E2 -18793.784} C_VEL
LIN {X 0,Y 250.432,Z 302.826,A -85,B 0,C 180,E1 -18795.371,E2 -18795.371} C_VEL
LIN {X 0,Y 249.469,Z 308.08,A -85,B 0,C 180,E1 -18796.976,E2 -18796.976} C_VEL
LIN {X 0,Y 248.622,Z 312.461,A -85,B 0,C 180,E1 -18798.588,E2 -18798.588} C_VEL
LIN {X 0,Y 247.736,Z 317.63,A -85,B 0,C 180,E1 -18801.024,E2 -18801.024} C_VEL
LIN {X 0,Y 247.16,Z 321.425,A -85,B 0,C 180,E1 -18803.469,E2 -18803.469} C_VEL
LIN {X 0,Y 246.969,Z 323.168,A -85,B 0,C 180,E1 -18805.103,E2 -18805.103} C_VEL
LIN {X 0,Y 246.879,Z 324.416,A -85,B 0,C 180,E1 -18806.737,E2 -18806.737} C_VEL
LIN {X 0,Y 246.87,Z 325.191,A -85,B 0,C 180,E1 -18808.369,E2 -18808.369} C_VEL
LIN {X 0,Y 246.899,Z 325.484,A -85,B 0,C 180,E1 -18810,E2 -18810} C_VEL
LIN {X 0,Y 246.87,Z 325.183,A -85,B 0,C 180,E1 -18811.632,E2 -18811.632} C_VEL
LIN {X 0,Y 246.879,Z 324.392,A -85,B 0,C 180,E1 -18813.264,E2 -18813.264} C_VEL
LIN {X 0,Y 246.989,Z 322.845,A -85,B 0,C 180,E1 -18815.182,E2 -18815.182} C_VEL
LIN {X 0,Y 247.304,Z 320.212,A -85,B 0,C 180,E1 -18817.348,E2 -18817.348} C_VEL
LIN {X 0,Y 247.678,Z 317.555,A -85,B 0,C 180,E1 -18818.979,E2 -18818.979} C_VEL
LIN {X 0,Y 248.616,Z 312.364,A -85,B 0,C 180,E1 -18821.413,E2 -18821.413} C_VEL
LIN {X 0,Y 249.933,Z 305.521,A -85,B 0,C 180,E1 -18823.829,E2 -18823.829} C_VEL
LIN {X 0,Y 251.318,Z 298.046,A -85,B 0,C 180,E1 -18825.823,E2 -18825.823} C_VEL
LIN {X 0,Y 252.706,Z 290.674,A -85,B 0,C 180,E1 -18827.396,E2 -18827.396} C_VEL
LIN {X 0,Y 254.095,Z 282.779,A -85,B 0,C 180,E1 -18828.756,E2 -18828.756} C_VEL
LIN {X 0,Y 255.319,Z 274.43,A -85,B 0,C 180,E1 -18829.916,E2 -18829.916} C_VEL
LIN {X 0,Y 256.573,Z 264.389,A -85,B 0,C 180,E1 -18831.005,E2 -18831.005} C_VEL
LIN {X 0,Y 257.716,Z 252.84,A -85,B 0,C 180,E1 -18831.869,E2 -18831.869} C_VEL
LIN {X 0,Y 258.425,Z 243.343,A -85,B 0,C 180,E1 -18832.336,E2 -18832.336} C_VEL
LIN {X 0,Y 259.245,Z 212.045,A -85,B 0,C 180,E1 -18833.24,E2 -18833.24} C_VEL
LIN {X 0,Y 259.193,Z 204.36,A -85,B 0,C 180,E1 -18833.472,E2 -18833.472} C_VEL
LIN {X 0,Y 255.778,Z 181.573,A -85,B 0,C 180,E1 -18834.488,E2 -18834.488} C_VEL
LIN {X 0,Y 253.558,Z 170.718,A -85,B 0,C 180,E1 -18835.047,E2 -18835.047} C_VEL
LIN {X 0,Y 251.793,Z 165.618,A -85,B 0,C 180,E1 -18835.45,E2 -18835.45} C_VEL
LIN {X 0,Y 250.676,Z 159.617,A -85,B 0,C 180,E1 -18838.009,E2 -18838.009} C_VEL
LIN {X 0,Y 249.05,Z 152.316,A -85,B 0,C 180,E1 -18841.513,E2 -18841.513} C_VEL
LIN {X 0,Y 249.05,Z 152.275,A -85,B 0,C 180,E1 -18845.08,E2 -18845.08} C_VEL
LIN {X 0,Y 249.028,Z 152.257,A -85,B 0,C 180,E1 -18848.381,E2 -18848.381} C_VEL
LIN {X 0,Y 249.002,Z 152.278,A -85,B 0,C 180,E1 -18852.791,E2 -18852.791} C_VEL
LIN {X 0,Y 249.01,Z 152.243,A -85,B 0,C 180,E1 -18857.362,E2 -18857.362} C_VEL
LIN {X 0,Y 249.026,Z 152.28,A -85,B 0,C 180,E1 -18861.62,E2 -18861.62} C_VEL
LIN {X 0,Y 249.045,Z 152.266,A -85,B 0,C 180,E1 -18865.64,E2 -18865.64} C_VEL
LIN {X 0,Y 249.053,Z 152.273,A -85,B 0,C 180,E1 -18869.474,E2 -18869.474} C_VEL
LIN {X 0,Y 249.076,Z 152.26,A -85,B 0,C 180,E1 -18873.163,E2 -18873.163} C_VEL
LIN {X 0,Y 249.081,Z 152.272,A -85,B 0,C 180,E1 -18876.733,E2 -18876.733} C_VEL
LIN {X 0,Y 249.112,Z 152.25,A -85,B 0,C 180,E1 -18880.212,E2 -18880.212} C_VEL
LIN {X 0,Y 249.244,Z 152.248,A -85,B 0,C 180,E1 -18883.622,E2 -18883.622} C_VEL
LIN {X 0,Y 249.247,Z 152.232,A -85,B 0,C 180,E1 -18888.616,E2 -18888.616} C_VEL
LIN {X 0,Y 249.457,Z 152.216,A -85,B 0,C 180,E1 -18891.902,E2 -18891.902} C_VEL
LIN {X 0,Y 249.297,Z 152.241,A -85,B 0,C 180,E1 -18895.149,E2 -18895.149} C_VEL
LIN {X 0,Y 249.677,Z 152.177,A -85,B 0,C 180,E1 -18898.387,E2 -18898.387} C_VEL
LIN {X 0,Y 249.677,Z 152.188,A -85,B 0,C 180,E1 -18901.613,E2 -18901.613} C_VEL
LIN {X 0,Y 249.453,Z 152.214,A -85,B 0,C 180,E1 -18906.733,E2 -18906.733} C_VEL
LIN {X 0,Y 249.391,Z 152.214,A -85,B 0,C 180,E1 -18909.735,E2 -18909.735} C_VEL
LIN {X 0,Y 249.208,Z 152.253,A -85,B 0,C 180,E1 -18914.703,E2 -18914.703} C_VEL
LIN {X 0,Y 249.142,Z 152.244,A -85,B 0,C 180,E1 -18918.077,E2 -18918.077} C_VEL
LIN {X 0,Y 249.09,Z 152.27,A -85,B 0,C 180,E1 -18921.518,E2 -18921.518} C_VEL
LIN {X 0,Y 249.132,Z 152.252,A -85,B 0,C 180,E1 -18925.482,E2 -18925.482} C_VEL
LIN {X 0,Y 249.085,Z 152.267,A -85,B 0,C 180,E1 -18928.993,E2 -18928.993} C_VEL
LIN {X 0,Y 249.033,Z 152.272,A -85,B 0,C 180,E1 -18932.426,E2 -18932.426} C_VEL
LIN {X 0,Y 249.05,Z 152.273,A -85,B 0,C 180,E1 -18936.342,E2 -18936.342} C_VEL
LIN {X 0,Y 249.008,Z 152.272,A -85,B 0,C 180,E1 -18940.478,E2 -18940.478} C_VEL
LIN {X 0,Y 248.997,Z 152.273,A -85,B 0,C 180,E1 -18944.881,E2 -18944.881} C_VEL
LIN {X 0,Y 249.011,Z 152.249,A -85,B 0,C 180,E1 -18947.361,E2 -18947.361} C_VEL
LIN {X 0,Y 249.04,Z 152.276,A -85,B 0,C 180,E1 -18951.622,E2 -18951.622} C_VEL
LIN {X 0,Y 249.061,Z 152.251,A -85,B 0,C 180,E1 -18955.642,E2 -18955.642} C_VEL
LIN {X 0,Y 249.054,Z 152.266,A -85,B 0,C 180,E1 -18959.473,E2 -18959.473} C_VEL
LIN {X 0,Y 249.167,Z 152.43,A -85,B 0,C 180,E1 -18962.035,E2 -18962.035} C_VEL
LIN {X 0,Y 250.171,Z 157.321,A -85,B 0,C 180,E1 -18964.366,E2 -18964.366} C_VEL
LIN {X 0,Y 250.841,Z 159.348,A -85,B 0,C 180,E1 -18964.611,E2 -18964.611} C_VEL
LIN {X 0,Y 256.491,Z 173.952,A -85,B 0,C 180,E1 -18965.654,E2 -18965.654} C_VEL
LIN {X 0,Y 258.378,Z 182.642,A -85,B 0,C 180,E1 -18966.104,E2 -18966.104} C_VEL
LIN {X 0,Y 259.797,Z 192.189,A -85,B 0,C 180,E1 -18966.526,E2 -18966.526} C_VEL
LIN {X 0,Y 258.6,Z 233.522,A -85,B 0,C 180,E1 -18967.678,E2 -18967.678} C_VEL
LIN {X 0,Y 258.09,Z 243.008,A -85,B 0,C 180,E1 -18968.135,E2 -18968.135} C_VEL
LIN {X 0,Y 257.334,Z 252.504,A -85,B 0,C 180,E1 -18968.809,E2 -18968.809} C_VEL
LIN {X 0,Y 256.087,Z 263.907,A -85,B 0,C 180,E1 -18969.937,E2 -18969.937} C_VEL
LIN {X 0,Y 254.618,Z 273.798,A -85,B 0,C 180,E1 -18971.284,E2 -18971.284} C_VEL
LIN {X 0,Y 253.305,Z 281.717,A -85,B 0,C 180,E1 -18972.646,E2 -18972.646} C_VEL
LIN {X 0,Y 252.305,Z 287.402,A -85,B 0,C 180,E1 -18973.826,E2 -18973.826} C_VEL
LIN {X 0,Y 251.094,Z 293.75,A -85,B 0,C 180,E1 -18975.409,E2 -18975.409} C_VEL
LIN {X 0,Y 250.047,Z 299.027,A -85,B 0,C 180,E1 -18977.005,E2 -18977.005} C_VEL
LIN {X 0,Y 249.131,Z 303.433,A -85,B 0,C 180,E1 -18978.611,E2 -18978.611} C_VEL
LIN {X 0,Y 248.223,Z 308.61,A -85,B 0,C 180,E1 -18981.041,E2 -18981.041} C_VEL
LIN {X 0,Y 247.699,Z 311.267,A -85,B 0,C 180,E1 -18982.664,E2 -18982.664} C_VEL
LIN {X 0,Y 247.519,Z 312.595,A -85,B 0,C 180,E1 -18983.608,E2 -18983.608} C_VEL
LIN {X 0,Y 247.231,Z 314.175,A -85,B 0,C 180,E1 -18985.107,E2 -18985.107} C_VEL
LIN {X 0,Y 247.059,Z 315.444,A -85,B 0,C 180,E1 -18986.738,E2 -18986.738} C_VEL
LIN {X 0,Y 246.926,Z 316.244,A -85,B 0,C 180,E1 -18988.369,E2 -18988.369} C_VEL
LIN {X 0,Y 246.927,Z 316.548,A -85,B 0,C 180,E1 -18990,E2 -18990} C_VEL
LIN {X 0,Y 246.925,Z 316.27,A -85,B 0,C 180,E1 -18991.631,E2 -18991.631} C_VEL
LIN {X 0,Y 247.056,Z 315.521,A -85,B 0,C 180,E1 -18993.261,E2 -18993.261} C_VEL
LIN {X 0,Y 247.414,Z 313.034,A -85,B 0,C 180,E1 -18996.171,E2 -18996.171} C_VEL
LIN {X 0,Y 247.895,Z 310.298,A -85,B 0,C 180,E1 -18998.149,E2 -18998.149} C_VEL
LIN {X 0,Y 248.766,Z 305.642,A -85,B 0,C 180,E1 -19000.581,E2 -19000.581} C_VEL
LIN {X 0,Y 249.787,Z 300.572,A -85,B 0,C 180,E1 -19002.594,E2 -19002.594} C_VEL
LIN {X 0,Y 250.759,Z 295.617,A -85,B 0,C 180,E1 -19004.195,E2 -19004.195} C_VEL
LIN {X 0,Y 251.954,Z 289.634,A -85,B 0,C 180,E1 -19005.781,E2 -19005.781} C_VEL
LIN {X 0,Y 253.204,Z 282.354,A -85,B 0,C 180,E1 -19007.36,E2 -19007.36} C_VEL
LIN {X 0,Y 254.566,Z 274.569,A -85,B 0,C 180,E1 -19008.719,E2 -19008.719} C_VEL
LIN {X 0,Y 255.611,Z 267.853,A -85,B 0,C 180,E1 -19009.682,E2 -19009.682} C_VEL
LIN {X 0,Y 256.696,Z 259.644,A -85,B 0,C 180,E1 -19010.64,E2 -19010.64} C_VEL
LIN {X 0,Y 257.684,Z 249.906,A -85,B 0,C 180,E1 -19011.517,E2 -19011.517} C_VEL
LIN {X 0,Y 258.43,Z 239.157,A -85,B 0,C 180,E1 -19012.21,E2 -19012.21} C_VEL
LIN {X 0,Y 258.955,Z 224.205,A -85,B 0,C 180,E1 -19012.741,E2 -19012.741} C_VEL
LIN {X 0,Y 259.709,Z 190.584,A -85,B 0,C 180,E1 -19013.662,E2 -19013.662} C_VEL
LIN {X 0,Y 257.104,Z 175.929,A -85,B 0,C 180,E1 -19014.358,E2 -19014.358} C_VEL
LIN {X 0,Y 253.21,Z 165.112,A -85,B 0,C 180,E1 -19015.091,E2 -19015.091} C_VEL
LIN {X 0,Y 250.3,Z 157.737,A -85,B 0,C 180,E1 -19015.681,E2 -19015.681} C_VEL
LIN {X 0,Y 250.119,Z 156.804,A -85,B 0,C 180,E1 -19015.952,E2 -19015.952} C_VEL
LIN {X 0,Y 249.135,Z 152.36,A -85,B 0,C 180,E1 -19018.197,E2 -19018.197} C_VEL
LIN {X 0,Y 249.036,Z 152.277,A -85,B 0,C 180,E1 -19022.424,E2 -19022.424} C_VEL
LIN {X 0,Y 249.069,Z 152.256,A -85,B 0,C 180,E1 -19026.338,E2 -19026.338} C_VEL
LIN {X 0,Y 249.026,Z 152.266,A -85,B 0,C 180,E1 -19030.474,E2 -19030.474} C_VEL
LIN {X 0,Y 248.993,Z 152.272,A -85,B 0,C 180,E1 -19034.881,E2 -19034.881} C_VEL
LIN {X 0,Y 249.015,Z 152.281,A -85,B 0,C 180,E1 -19037.362,E2 -19037.362} C_VEL
LIN {X 0,Y 249.043,Z 152.275,A -85,B 0,C 180,E1 -19042.2,E2 -19042.2} C_VEL
LIN {X 0,Y 249.043,Z 152.264,A -85,B 0,C 180,E1 -19045.639,E2 -19045.639} C_VEL
LIN {X 0,Y 249.051,Z 152.275,A -85,B 0,C 180,E1 -19049.473,E2 -19049.473} C_VEL
LIN {X 0,Y 249.072,Z 152.257,A -85,B 0,C 180,E1 -19053.162,E2 -19053.162} C_VEL
LIN {X 0,Y 249.079,Z 152.27,A -85,B 0,C 180,E1 -19056.732,E2 -19056.732} C_VEL
LIN {X 0,Y 249.11,Z 152.259,A -85,B 0,C 180,E1 -19060.211,E2 -19060.211} C_VEL
LIN {X 0,Y 249.241,Z 152.242,A -85,B 0,C 180,E1 -19063.622,E2 -19063.622} C_VEL
LIN {X 0,Y 249.253,Z 152.242,A -85,B 0,C 180,E1 -19068.616,E2 -19068.616} C_VEL
LIN {X 0,Y 249.48,Z 152.202,A -85,B 0,C 180,E1 -19071.903,E2 -19071.903} C_VEL
LIN {X 0,Y 249.436,Z 152.224,A -85,B 0,C 180,E1 -19076.769,E2 -19076.769} C_VEL
LIN {X 0,Y 249.727,Z 152.172,A -85,B 0,C 180,E1 -19080,E2 -19080} C_VEL
LIN {X 0,Y 249.435,Z 152.219,A -85,B 0,C 180,E1 -19083.23,E2 -19083.23} C_VEL
LIN {X 0,Y 249.481,Z 152.213,A -85,B 0,C 180,E1 -19088.097,E2 -19088.097} C_VEL
LIN {X 0,Y 249.252,Z 152.232,A -85,B 0,C 180,E1 -19091.383,E2 -19091.383} C_VEL
LIN {X 0,Y 249.213,Z 152.25,A -85,B 0,C 180,E1 -19095.994,E2 -19095.994} C_VEL
LIN {X 0,Y 248.93,Z 152.288,A -85,B 0,C 180,E1 -19096.895,E2 -19096.895} C_VEL
LIN {X 0,Y 247.573,Z 152.457,A -85,B 0,C 180,E1 -19098.226,E2 -19098.226} C_VEL
LIN {X 0,Y 243.133,Z 153.005,A -85,B 0,C 180,E1 -19101.325,E2 -19101.325} C_VEL
LIN {X 0,Y 242.078,Z 153.141,A -85,B 0,C 180,E1 -19102.715,E2 -19102.715} C_VEL
LIN {X 0,Y 242.007,Z 153.146,A -85,B 0,C 180,E1 -19103.187,E2 -19103.187} C_VEL
LIN {X 0,Y 242.065,Z 153.138,A -85,B 0,C 180,E1 -19105.838,E2 -19105.838} C_VEL
LIN {X 0,Y 242.029,Z 153.146,A -85,B 0,C 180,E1 -19109.58,E2 -19109.58} C_VEL
LIN {X 0,Y 241.979,Z 153.149,A -85,B 0,C 180,E1 -19113.493,E2 -19113.493} C_VEL
LIN {X 0,Y 241.988,Z 153.154,A -85,B 0,C 180,E1 -19117.582,E2 -19117.582} C_VEL
LIN {X 0,Y 241.932,Z 153.13,A -85,B 0,C 180,E1 -19121.923,E2 -19121.923} C_VEL
LIN {X 0,Y 241.924,Z 153.155,A -85,B 0,C 180,E1 -19126.574,E2 -19126.574} C_VEL
LIN {X 0,Y 241.955,Z 153.144,A -85,B 0,C 180,E1 -19130.281,E2 -19130.281} C_VEL
LIN {X 0,Y 241.991,Z 153.156,A -85,B 0,C 180,E1 -19134.49,E2 -19134.49} C_VEL
LIN {X 0,Y 242.024,Z 153.339,A -85,B 0,C 180,E1 -19138.012,E2 -19138.012} C_VEL
LIN {X 0,Y 243.659,Z 160.638,A -85,B 0,C 180,E1 -19141.581,E2 -19141.581} C_VEL
LIN {X 0,Y 244.589,Z 165.485,A -85,B 0,C 180,E1 -19143.699,E2 -19143.699} C_VEL
LIN {X 0,Y 248.036,Z 175.193,A -85,B 0,C 180,E1 -19144.453,E2 -19144.453} C_VEL
LIN {X 0,Y 251.976,Z 199.416,A -85,B 0,C 180,E1 -19145.622,E2 -19145.622} C_VEL
LIN {X 0,Y 252.91,Z 208.196,A -85,B 0,C 180,E1 -19145.985,E2 -19145.985} C_VEL
LIN {X 0,Y 251.881,Z 243.179,A -85,B 0,C 180,E1 -19147.007,E2 -19147.007} C_VEL
LIN {X 0,Y 251.057,Z 254.63,A -85,B 0,C 180,E1 -19147.604,E2 -19147.604} C_VEL
LIN {X 0,Y 249.823,Z 265.928,A -85,B 0,C 180,E1 -19148.549,E2 -19148.549} C_VEL
LIN {X 0,Y 248.653,Z 274.603,A -85,B 0,C 180,E1 -19149.527,E2 -19149.527} C_VEL
LIN {X 0,Y 247.398,Z 282.895,A -85,B 0,C 180,E1 -19150.717,E2 -19150.717} C_VEL
LIN {X 0,Y 245.908,Z 290.743,A -85,B 0,C 180,E1 -19152.108,E2 -19152.108} C_VEL
LIN {X 0,Y 244.496,Z 298.085,A -85,B 0,C 180,E1 -19153.725,E2 -19153.725} C_VEL
LIN {X 0,Y 243.041,Z 305.535,A -85,B 0,C 180,E1 -19155.772,E2 -19155.772} C_VEL
LIN {X 0,Y 241.658,Z 312.334,A -85,B 0,C 180,E1 -19158.254,E2 -19158.254} C_VEL
LIN {X 0,Y 240.714,Z 317.502,A -85,B 0,C 180,E1 -19160.76,E2 -19160.76} C_VEL
LIN {X 0,Y 240.087,Z 321.297,A -85,B 0,C 180,E1 -19163.276,E2 -19163.276} C_VEL
LIN {X 0,Y 239.879,Z 323.04,A -85,B 0,C 180,E1 -19164.958,E2 -19164.958} C_VEL
LIN {X 0,Y 239.788,Z 324.288,A -85,B 0,C 180,E1 -19166.64,E2 -19166.64} C_VEL
LIN {X 0,Y 239.785,Z 325.063,A -85,B 0,C 180,E1 -19168.321,E2 -19168.321} C_VEL
LIN {X 0,Y 239.811,Z 325.355,A -85,B 0,C 180,E1 -19170,E2 -19170} C_VEL
LIN {X 0,Y 239.785,Z 325.055,A -85,B 0,C 180,E1 -19171.68,E2 -19171.68} C_VEL
LIN {X 0,Y 239.788,Z 324.263,A -85,B 0,C 180,E1 -19173.361,E2 -19173.361} C_VEL
LIN {X 0,Y 239.88,Z 322.999,A -85,B 0,C 180,E1 -19175.043,E2 -19175.043} C_VEL
LIN {X 0,Y 240.239,Z 320.082,A -85,B 0,C 180,E1 -19177.565,E2 -19177.565} C_VEL
LIN {X 0,Y 240.668,Z 317.425,A -85,B 0,C 180,E1 -19179.243,E2 -19179.243} C_VEL
LIN {X 0,Y 241.653,Z 312.234,A -85,B 0,C 180,E1 -19181.747,E2 -19181.747} C_VEL
LIN {X 0,Y 243.026,Z 305.391,A -85,B 0,C 180,E1 -19184.23,E2 -19184.23} C_VEL
LIN {X 0,Y 244.491,Z 297.914,A -85,B 0,C 180,E1 -19186.277,E2 -19186.277} C_VEL
LIN {X 0,Y 245.929,Z 290.542,A -85,B 0,C 180,E1 -19187.891,E2 -19187.891} C_VEL
LIN {X 0,Y 247.386,Z 282.647,A -85,B 0,C 180,E1 -19189.285,E2 -19189.285} C_VEL
LIN {X 0,Y 248.663,Z 274.297,A -85,B 0,C 180,E1 -19190.473,E2 -19190.473} C_VEL
LIN {X 0,Y 250.095,Z 263.263,A -85,B 0,C 180,E1 -19191.679,E2 -19191.679} C_VEL
LIN {X 0,Y 251.178,Z 252.227,A -85,B 0,C 180,E1 -19192.5,E2 -19192.5} C_VEL
LIN {X 0,Y 251.904,Z 242.878,A -85,B 0,C 180,E1 -19192.96,E2 -19192.96} C_VEL
LIN {X 0,Y 252.779,Z 205.876,A -85,B 0,C 180,E1 -19194.054,E2 -19194.054} C_VEL
LIN {X 0,Y 249.335,Z 182.756,A -85,B 0,C 180,E1 -19195.123,E2 -19195.123} C_VEL
LIN {X 0,Y 247.425,Z 173.282,A -85,B 0,C 180,E1 -19195.627,E2 -19195.627} C_VEL
LIN {X 0,Y 244.593,Z 165.444,A -85,B 0,C 180,E1 -19196.26,E2 -19196.26} C_VEL
LIN {X 0,Y 243.433,Z 159.472,A -85,B 0,C 180,E1 -19198.92,E2 -19198.92} C_VEL
LIN {X 0,Y 242,Z 153.176,A -85,B 0,C 180,E1 -19202.088,E2 -19202.088} C_VEL
LIN {X 0,Y 242.006,Z 153.154,A -85,B 0,C 180,E1 -19205.597,E2 -19205.597} C_VEL
LIN {X 0,Y 241.957,Z 153.145,A -85,B 0,C 180,E1 -19209.719,E2 -19209.719} C_VEL
LIN {X 0,Y 241.919,Z 153.147,A -85,B 0,C 180,E1 -19214.205,E2 -19214.205} C_VEL
LIN {X 0,Y 241.934,Z 153.13,A -85,B 0,C 180,E1 -19218.077,E2 -19218.077} C_VEL
LIN {X 0,Y 241.99,Z 153.154,A -85,B 0,C 180,E1 -19222.419,E2 -19222.419} C_VEL
LIN {X 0,Y 241.982,Z 153.149,A -85,B 0,C 180,E1 -19226.508,E2 -19226.508} C_VEL
LIN {X 0,Y 242.038,Z 153.142,A -85,B 0,C 180,E1 -19230.587,E2 -19230.587} C_VEL
LIN {X 0,Y 242.069,Z 153.138,A -85,B 0,C 180,E1 -19234.183,E2 -19234.183} C_VEL
LIN {X 0,Y 242.055,Z 153.141,A -85,B 0,C 180,E1 -19238.297,E2 -19238.297} C_VEL
LIN {X 0,Y 242.165,Z 153.131,A -85,B 0,C 180,E1 -19243.278,E2 -19243.278} C_VEL
LIN {X 0,Y 242.183,Z 153.114,A -85,B 0,C 180,E1 -19248.28,E2 -19248.28} C_VEL
LIN {X 0,Y 242.402,Z 153.094,A -85,B 0,C 180,E1 -19251.665,E2 -19251.665} C_VEL
LIN {X 0,Y 242.258,Z 153.119,A -85,B 0,C 180,E1 -19255.007,E2 -19255.007} C_VEL
LIN {X 0,Y 242.638,Z 153.053,A -85,B 0,C 180,E1 -19258.34,E2 -19258.34} C_VEL
LIN {X 0,Y 242.638,Z 153.065,A -85,B 0,C 180,E1 -19261.66,E2 -19261.66} C_VEL
LIN {X 0,Y 242.432,Z 153.09,A -85,B 0,C 180,E1 -19266.709,E2 -19266.709} C_VEL
LIN {X 0,Y 242.316,Z 153.096,A -85,B 0,C 180,E1 -19270.022,E2 -19270.022} C_VEL
LIN {X 0,Y 242.17,Z 153.131,A -85,B 0,C 180,E1 -19275.141,E2 -19275.141} C_VEL
LIN {X 0,Y 242.075,Z 153.123,A -85,B 0,C 180,E1 -19278.624,E2 -19278.624} C_VEL
LIN {X 0,Y 242.015,Z 153.149,A -85,B 0,C 180,E1 -19282.18,E2 -19282.18} C_VEL
LIN {X 0,Y 242.069,Z 153.13,A -85,B 0,C 180,E1 -19285.838,E2 -19285.838} C_VEL
LIN {X 0,Y 242.032,Z 153.148,A -85,B 0,C 180,E1 -19289.58,E2 -19289.58} C_VEL
LIN {X 0,Y 241.983,Z 153.141,A -85,B 0,C 180,E1 -19293.493,E2 -19293.493} C_VEL
LIN {X 0,Y 241.991,Z 153.153,A -85,B 0,C 180,E1 -19297.582,E2 -19297.582} C_VEL
LIN {X 0,Y 241.939,Z 153.159,A -85,B 0,C 180,E1 -19301.922,E2 -19301.922} C_VEL
LIN {X 0,Y 241.929,Z 153.134,A -85,B 0,C 180,E1 -19306.573,E2 -19306.573} C_VEL
LIN {X 0,Y 241.974,Z 153.149,A -85,B 0,C 180,E1 -19310.284,E2 -19310.284} C_VEL
LIN {X 0,Y 242.039,Z 153.125,A -85,B 0,C 180,E1 -19314.497,E2 -19314.497} C_VEL
LIN {X 0,Y 241.978,Z 153.155,A -85,B 0,C 180,E1 -19318.48,E2 -19318.48} C_VEL
LIN {X 0,Y 242.094,Z 153.307,A -85,B 0,C 180,E1 -19321.498,E2 -19321.498} C_VEL
LIN {X 0,Y 243.032,Z 157.568,A -85,B 0,C 180,E1 -19323.578,E2 -19323.578} C_VEL
LIN {X 0,Y 243.994,Z 160.21,A -85,B 0,C 180,E1 -19323.868,E2 -19323.868} C_VEL
LIN {X 0,Y 250.027,Z 175.598,A -85,B 0,C 180,E1 -19325.028,E2 -19325.028} C_VEL
LIN {X 0,Y 251.501,Z 181.36,A -85,B 0,C 180,E1 -19325.363,E2 -19325.363} C_VEL
LIN {X 0,Y 253.308,Z 192.22,A -85,B 0,C 180,E1 -19325.883,E2 -19325.883} C_VEL
LIN {X 0,Y 252.028,Z 234.248,A -85,B 0,C 180,E1 -19327.087,E2 -19327.087} C_VEL
LIN {X 0,Y 251.42,Z 244.659,A -85,B 0,C 180,E1 -19327.622,E2 -19327.622} C_VEL
LIN {X 0,Y 250.33,Z 256.733,A -85,B 0,C 180,E1 -19328.594,E2 -19328.594} C_VEL
LIN {X 0,Y 249.17,Z 265.545,A -85,B 0,C 180,E1 -19329.571,E2 -19329.571} C_VEL
LIN {X 0,Y 247.92,Z 273.93,A -85,B 0,C 180,E1 -19330.759,E2 -19330.759} C_VEL
LIN {X 0,Y 246.537,Z 281.848,A -85,B 0,C 180,E1 -19332.154,E2 -19332.154} C_VEL
LIN {X 0,Y 245.492,Z 287.533,A -85,B 0,C 180,E1 -19333.364,E2 -19333.364} C_VEL
LIN {X 0,Y 244.243,Z 293.881,A -85,B 0,C 180,E1 -19334.991,E2 -19334.991} C_VEL
LIN {X 0,Y 243.13,Z 299.158,A -85,B 0,C 180,E1 -19336.629,E2 -19336.629} C_VEL
LIN {X 0,Y 242.191,Z 303.562,A -85,B 0,C 180,E1 -19338.28,E2 -19338.28} C_VEL
LIN {X 0,Y 241.197,Z 308.74,A -85,B 0,C 180,E1 -19340.778,E2 -19340.778} C_VEL
LIN {X 0,Y 240.65,Z 311.397,A -85,B 0,C 180,E1 -19342.448,E2 -19342.448} C_VEL
LIN {X 0,Y 240.406,Z 313.068,A -85,B 0,C 180,E1 -19343.697,E2 -19343.697} C_VEL
LIN {X 0,Y 239.966,Z 315.572,A -85,B 0,C 180,E1 -19346.642,E2 -19346.642} C_VEL
LIN {X 0,Y 239.843,Z 316.372,A -85,B 0,C 180,E1 -19348.32,E2 -19348.32} C_VEL
LIN {X 0,Y 239.838,Z 316.676,A -85,B 0,C 180,E1 -19350,E2 -19350} C_VEL
LIN {X 0,Y 239.842,Z 316.398,A -85,B 0,C 180,E1 -19351.679,E2 -19351.679} C_VEL
LIN {X 0,Y 239.963,Z 315.649,A -85,B 0,C 180,E1 -19353.358,E2 -19353.358} C_VEL
LIN {X 0,Y 240.313,Z 313.412,A -85,B 0,C 180,E1 -19356.1,E2 -19356.1} C_VEL
LIN {X 0,Y 240.875,Z 310.425,A -85,B 0,C 180,E1 -19358.388,E2 -19358.388} C_VEL
LIN {X 0,Y 241.78,Z 305.769,A -85,B 0,C 180,E1 -19360.891,E2 -19360.891} C_VEL
LIN {X 0,Y 242.846,Z 300.699,A -85,B 0,C 180,E1 -19362.96,E2 -19362.96} C_VEL
LIN {X 0,Y 243.889,Z 295.743,A -85,B 0,C 180,E1 -19364.604,E2 -19364.604} C_VEL
LIN {X 0,Y 245.132,Z 289.76,A -85,B 0,C 180,E1 -19366.232,E2 -19366.232} C_VEL
LIN {X 0,Y 246.45,Z 282.479,A -85,B 0,C 180,E1 -19367.851,E2 -19367.851} C_VEL
LIN {X 0,Y 247.858,Z 274.693,A -85,B 0,C 180,E1 -19369.246,E2 -19369.246} C_VEL
LIN {X 0,Y 248.937,Z 267.976,A -85,B 0,C 180,E1 -19370.233,E2 -19370.233} C_VEL
LIN {X 0,Y 250.066,Z 259.766,A -85,B 0,C 180,E1 -19371.213,E2 -19371.213} C_VEL
LIN {X 0,Y 251.078,Z 250.314,A -85,B 0,C 180,E1 -19372.086,E2 -19372.086} C_VEL
LIN {X 0,Y 251.845,Z 239.86,A -85,B 0,C 180,E1 -19372.784,E2 -19372.784} C_VEL
LIN {X 0,Y 252.36,Z 226.663,A -85,B 0,C 180,E1 -19373.298,E2 -19373.298} C_VEL
LIN {X 0,Y 253.241,Z 191.676,A -85,B 0,C 180,E1 -19374.275,E2 -19374.275} C_VEL
LIN {X 0,Y 250.675,Z 177.426,A -85,B 0,C 180,E1 -19374.982,E2 -19374.982} C_VEL
LIN {X 0,Y 245.228,Z 163.125,A -85,B 0,C 180,E1 -19376.035,E2 -19376.035} C_VEL
LIN {X 0,Y 243.109,Z 157.889,A -85,B 0,C 180,E1 -19376.496,E2 -19376.496} C_VEL
LIN {X 0,Y 242.855,Z 156.827,A -85,B 0,C 180,E1 -19376.842,E2 -19376.842} C_VEL
LIN {X 0,Y 242.064,Z 153.252,A -85,B 0,C 180,E1 -19378.721,E2 -19378.721} C_VEL
LIN {X 0,Y 241.991,Z 153.141,A -85,B 0,C 180,E1 -19383.49,E2 -19383.49} C_VEL
LIN {X 0,Y 242.002,Z 153.149,A -85,B 0,C 180,E1 -19387.579,E2 -19387.579} C_VEL
LIN {X 0,Y 241.938,Z 153.127,A -85,B 0,C 180,E1 -19391.921,E2 -19391.921} C_VEL
LIN {X 0,Y 241.932,Z 153.161,A -85,B 0,C 180,E1 -19396.571,E2 -19396.571} C_VEL
LIN {X 0,Y 241.956,Z 153.149,A -85,B 0,C 180,E1 -19400.28,E2 -19400.28} C_VEL
LIN {X 0,Y 241.987,Z 153.152,A -85,B 0,C 180,E1 -19404.489,E2 -19404.489} C_VEL
LIN {X 0,Y 241.974,Z 153.153,A -85,B 0,C 180,E1 -19408.479,E2 -19408.479} C_VEL
LIN {X 0,Y 242.008,Z 153.143,A -85,B 0,C 180,E1 -19412.312,E2 -19412.312} C_VEL
LIN {X 0,Y 242.056,Z 153.141,A -85,B 0,C 180,E1 -19416.016,E2 -19416.016} C_VEL
LIN {X 0,Y 242.037,Z 153.141,A -85,B 0,C 180,E1 -19419.608,E2 -19419.608} C_VEL
LIN {X 0,Y 242.162,Z 153.121,A -85,B 0,C 180,E1 -19423.278,E2 -19423.278} C_VEL
LIN {X 0,Y 242.186,Z 153.125,A -85,B 0,C 180,E1 -19428.28,E2 -19428.28} C_VEL
LIN {X 0,Y 242.427,Z 153.079,A -85,B 0,C 180,E1 -19431.665,E2 -19431.665} C_VEL
LIN {X 0,Y 242.26,Z 153.119,A -85,B 0,C 180,E1 -19435.007,E2 -19435.007} C_VEL
LIN {X 0,Y 242.636,Z 153.065,A -85,B 0,C 180,E1 -19438.34,E2 -19438.34} C_VEL
LIN {X 0,Y 242.635,Z 153.053,A -85,B 0,C 180,E1 -19441.66,E2 -19441.66} C_VEL
LIN {X 0,Y 242.433,Z 153.096,A -85,B 0,C 180,E1 -19446.659,E2 -19446.659} C_VEL
LIN {X 0,Y 242.313,Z 153.092,A -85,B 0,C 180,E1 -19450.022,E2 -19450.022} C_VEL
LIN {X 0,Y 242.165,Z 153.133,A -85,B 0,C 180,E1 -19455.141,E2 -19455.141} C_VEL
LIN {X 0,Y 242.072,Z 153.13,A -85,B 0,C 180,E1 -19458.624,E2 -19458.624} C_VEL
LIN {X 0,Y 242.007,Z 153.146,A -85,B 0,C 180,E1 -19463.187,E2 -19463.187} C_VEL
LIN {X 0,Y 241.385,Z 153.23,A -85,B 0,C 180,E1 -19464.575,E2 -19464.575} C_VEL
LIN {X 0,Y 238.566,Z 153.589,A -85,B 0,C 180,E1 -19466.839,E2 -19466.839} C_VEL
LIN {X 0,Y 236.122,Z 153.894,A -85,B 0,C 180,E1 -19468.683,E2 -19468.683} C_VEL
LIN {X 0,Y 235.035,Z 154.023,A -85,B 0,C 180,E1 -19470.114,E2 -19470.114} C_VEL
LIN {X 0,Y 234.928,Z 154.032,A -85,B 0,C 180,E1 -19470.6,E2 -19470.6} C_VEL
LIN {X 0,Y 234.929,Z 154.022,A -85,B 0,C 180,E1 -19474.638,E2 -19474.638} C_VEL
LIN {X 0,Y 234.94,Z 154.03,A -85,B 0,C 180,E1 -19478.945,E2 -19478.945} C_VEL
LIN {X 0,Y 234.876,Z 153.997,A -85,B 0,C 180,E1 -19483.488,E2 -19483.488} C_VEL
LIN {X 0,Y 234.876,Z 154.032,A -85,B 0,C 180,E1 -19486.512,E2 -19486.512} C_VEL
LIN {X 0,Y 234.917,Z 154.013,A -85,B 0,C 180,E1 -19491.079,E2 -19491.079} C_VEL
LIN {X 0,Y 234.932,Z 154.029,A -85,B 0,C 180,E1 -19495.363,E2 -19495.363} C_VEL
LIN {X 0,Y 234.974,Z 154.218,A -85,B 0,C 180,E1 -19497.428,E2 -19497.428} C_VEL
LIN {X 0,Y 236.842,Z 162.598,A -85,B 0,C 180,E1 -19501.655,E2 -19501.655} C_VEL
LIN {X 0,Y 237.337,Z 165.311,A -85,B 0,C 180,E1 -19502.824,E2 -19502.824} C_VEL
LIN {X 0,Y 241.222,Z 175.373,A -85,B 0,C 180,E1 -19503.686,E2 -19503.686} C_VEL
LIN {X 0,Y 242.871,Z 183.081,A -85,B 0,C 180,E1 -19504.126,E2 -19504.126} C_VEL
LIN {X 0,Y 246.248,Z 205.864,A -85,B 0,C 180,E1 -19505.223,E2 -19505.223} C_VEL
LIN {X 0,Y 246.259,Z 212.976,A -85,B 0,C 180,E1 -19505.448,E2 -19505.448} C_VEL
LIN {X 0,Y 245.368,Z 243.067,A -85,B 0,C 180,E1 -19506.36,E2 -19506.36} C_VEL
LIN {X 0,Y 244.503,Z 254.517,A -85,B 0,C 180,E1 -19506.97,E2 -19506.97} C_VEL
LIN {X 0,Y 243.239,Z 265.805,A -85,B 0,C 180,E1 -19507.938,E2 -19507.938} C_VEL
LIN {X 0,Y 242.006,Z 274.479,A -85,B 0,C 180,E1 -19508.939,E2 -19508.939} C_VEL
LIN {X 0,Y 240.711,Z 282.77,A -85,B 0,C 180,E1 -19510.159,E2 -19510.159} C_VEL
LIN {X 0,Y 239.17,Z 290.618,A -85,B 0,C 180,E1 -19511.586,E2 -19511.586} C_VEL
LIN {X 0,Y 237.69,Z 297.959,A -85,B 0,C 180,E1 -19513.245,E2 -19513.245} C_VEL
LIN {X 0,Y 236.156,Z 305.408,A -85,B 0,C 180,E1 -19515.348,E2 -19515.348} C_VEL
LIN {X 0,Y 234.697,Z 312.206,A -85,B 0,C 180,E1 -19517.901,E2 -19517.901} C_VEL
LIN {X 0,Y 233.686,Z 317.375,A -85,B 0,C 180,E1 -19520.479,E2 -19520.479} C_VEL
LIN {X 0,Y 233.021,Z 321.169,A -85,B 0,C 180,E1 -19523.071,E2 -19523.071} C_VEL
LIN {X 0,Y 232.777,Z 323.18,A -85,B 0,C 180,E1 -19525.09,E2 -19525.09} C_VEL
LIN {X 0,Y 232.683,Z 324.934,A -85,B 0,C 180,E1 -19528.27,E2 -19528.27} C_VEL
LIN {X 0,Y 232.725,Z 325.227,A -85,B 0,C 180,E1 -19530,E2 -19530} C_VEL
LIN {X 0,Y 232.683,Z 324.926,A -85,B 0,C 180,E1 -19531.731,E2 -19531.731} C_VEL
LIN {X 0,Y 232.758,Z 323.191,A -85,B 0,C 180,E1 -19534.854,E2 -19534.854} C_VEL
LIN {X 0,Y 233.051,Z 321.109,A -85,B 0,C 180,E1 -19536.929,E2 -19536.929} C_VEL
LIN {X 0,Y 233.649,Z 317.295,A -85,B 0,C 180,E1 -19539.523,E2 -19539.523} C_VEL
LIN {X 0,Y 234.693,Z 312.104,A -85,B 0,C 180,E1 -19542.1,E2 -19542.1} C_VEL
LIN {X 0,Y 236.141,Z 305.26,A -85,B 0,C 180,E1 -19544.654,E2 -19544.654} C_VEL
LIN {X 0,Y 237.688,Z 297.784,A -85,B 0,C 180,E1 -19546.756,E2 -19546.756} C_VEL
LIN {X 0,Y 239.188,Z 290.411,A -85,B 0,C 180,E1 -19548.413,E2 -19548.413} C_VEL
LIN {X 0,Y 240.686,Z 282.514,A -85,B 0,C 180,E1 -19549.844,E2 -19549.844} C_VEL
LIN {X 0,Y 242.032,Z 274.164,A -85,B 0,C 180,E1 -19551.06,E2 -19551.06} C_VEL
LIN {X 0,Y 243.431,Z 263.847,A -85,B 0,C 180,E1 -19552.228,E2 -19552.228} C_VEL
LIN {X 0,Y 244.598,Z 252.551,A -85,B 0,C 180,E1 -19553.109,E2 -19553.109} C_VEL
LIN {X 0,Y 245.386,Z 242.942,A -85,B 0,C 180,E1 -19553.597,E2 -19553.597} C_VEL
LIN {X 0,Y 246.309,Z 210.951,A -85,B 0,C 180,E1 -19554.564,E2 -19554.564} C_VEL
LIN {X 0,Y 246.186,Z 205.586,A -85,B 0,C 180,E1 -19554.745,E2 -19554.745} C_VEL
LIN {X 0,Y 242.231,Z 179.734,A -85,B 0,C 180,E1 -19556.006,E2 -19556.006} C_VEL
LIN {X 0,Y 241.127,Z 175.267,A -85,B 0,C 180,E1 -19556.278,E2 -19556.278} C_VEL
LIN {X 0,Y 237.413,Z 165.59,A -85,B 0,C 180,E1 -19557.074,E2 -19557.074} C_VEL
LIN {X 0,Y 237.046,Z 163.867,A -85,B 0,C 180,E1 -19557.685,E2 -19557.685} C_VEL
LIN {X 0,Y 235.632,Z 157.214,A -85,B 0,C 180,E1 -19560.964,E2 -19560.964} C_VEL
LIN {X 0,Y 234.959,Z 154.056,A -85,B 0,C 180,E1 -19562.671,E2 -19562.671} C_VEL
LIN {X 0,Y 234.929,Z 154.019,A -85,B 0,C 180,E1 -19566.749,E2 -19566.749} C_VEL
LIN {X 0,Y 234.943,Z 154.011,A -85,B 0,C 180,E1 -19568.945,E2 -19568.945} C_VEL
LIN {X 0,Y 234.879,Z 154.03,A -85,B 0,C 180,E1 -19573.488,E2 -19573.488} C_VEL
LIN {X 0,Y 234.878,Z 153.996,A -85,B 0,C 180,E1 -19576.512,E2 -19576.512} C_VEL
LIN {X 0,Y 234.919,Z 154.033,A -85,B 0,C 180,E1 -19581.079,E2 -19581.079} C_VEL
LIN {X 0,Y 234.931,Z 154.021,A -85,B 0,C 180,E1 -19585.362,E2 -19585.362} C_VEL
LIN {X 0,Y 234.933,Z 154.032,A -85,B 0,C 180,E1 -19589.433,E2 -19589.433} C_VEL
LIN {X 0,Y 234.996,Z 154.018,A -85,B 0,C 180,E1 -19593.794,E2 -19593.794} C_VEL
LIN {X 0,Y 235.013,Z 154.01,A -85,B 0,C 180,E1 -19598.97,E2 -19598.97} C_VEL
LIN {X 0,Y 235.098,Z 154.009,A -85,B 0,C 180,E1 -19603.06,E2 -19603.06} C_VEL
LIN {X 0,Y 235.117,Z 153.997,A -85,B 0,C 180,E1 -19607.922,E2 -19607.922} C_VEL
LIN {X 0,Y 235.333,Z 153.973,A -85,B 0,C 180,E1 -19611.413,E2 -19611.413} C_VEL
LIN {X 0,Y 235.395,Z 153.973,A -85,B 0,C 180,E1 -19613.141,E2 -19613.141} C_VEL
LIN {X 0,Y 235.597,Z 153.929,A -85,B 0,C 180,E1 -19618.291,E2 -19618.291} C_VEL
LIN {X 0,Y 235.598,Z 153.942,A -85,B 0,C 180,E1 -19621.71,E2 -19621.71} C_VEL
LIN {X 0,Y 235.407,Z 153.966,A -85,B 0,C 180,E1 -19626.859,E2 -19626.859} C_VEL
LIN {X 0,Y 235.24,Z 153.98,A -85,B 0,C 180,E1 -19630.327,E2 -19630.327} C_VEL
LIN {X 0,Y 235.116,Z 154.004,A -85,B 0,C 180,E1 -19635.606,E2 -19635.606} C_VEL
LIN {X 0,Y 235.011,Z 154.005,A -85,B 0,C 180,E1 -19639.206,E2 -19639.206} C_VEL
LIN {X 0,Y 234.963,Z 154.029,A -85,B 0,C 180,E1 -19642.883,E2 -19642.883} C_VEL
LIN {X 0,Y 234.972,Z 154.011,A -85,B 0,C 180,E1 -19646.657,E2 -19646.657} C_VEL
LIN {X 0,Y 234.934,Z 154.034,A -85,B 0,C 180,E1 -19650.568,E2 -19650.568} C_VEL
LIN {X 0,Y 234.933,Z 154.021,A -85,B 0,C 180,E1 -19654.638,E2 -19654.638} C_VEL
LIN {X 0,Y 234.944,Z 154.025,A -85,B 0,C 180,E1 -19658.944,E2 -19658.944} C_VEL
LIN {X 0,Y 234.887,Z 154.039,A -85,B 0,C 180,E1 -19663.486,E2 -19663.486} C_VEL
LIN {X 0,Y 234.882,Z 154.01,A -85,B 0,C 180,E1 -19666.512,E2 -19666.512} C_VEL
LIN {X 0,Y 234.957,Z 154.03,A -85,B 0,C 180,E1 -19671.086,E2 -19671.086} C_VEL
LIN {X 0,Y 234.962,Z 154.004,A -85,B 0,C 180,E1 -19675.367,E2 -19675.367} C_VEL
LIN {X 0,Y 234.972,Z 154.018,A -85,B 0,C 180,E1 -19680.157,E2 -19680.157} C_VEL
LIN {X 0,Y 235.059,Z 154.307,A -85,B 0,C 180,E1 -19681.016,E2 -19681.016} C_VEL
LIN {X 0,Y 235.817,Z 157.776,A -85,B 0,C 180,E1 -19682.718,E2 -19682.718} C_VEL
LIN {X 0,Y 237.368,Z 161.502,A -85,B 0,C 180,E1 -19683.119,E2 -19683.119} C_VEL
LIN {X 0,Y 243.852,Z 177.897,A -85,B 0,C 180,E1 -19684.419,E2 -19684.419} C_VEL
LIN {X 0,Y 245.217,Z 183.334,A -85,B 0,C 180,E1 -19684.746,E2 -19684.746} C_VEL
LIN {X 0,Y 246.825,Z 193.417,A -85,B 0,C 180,E1 -19685.24,E2 -19685.24} C_VEL
LIN {X 0,Y 245.553,Z 233.837,A -85,B 0,C 180,E1 -19686.423,E2 -19686.423} C_VEL
LIN {X 0,Y 244.978,Z 243.33,A -85,B 0,C 180,E1 -19686.902,E2 -19686.902} C_VEL
LIN {X 0,Y 244.127,Z 253.24,A -85,B 0,C 180,E1 -19687.645,E2 -19687.645} C_VEL
LIN {X 0,Y 242.832,Z 264.174,A -85,B 0,C 180,E1 -19688.791,E2 -19688.791} C_VEL
LIN {X 0,Y 241.248,Z 274.062,A -85,B 0,C 180,E1 -19690.205,E2 -19690.205} C_VEL
LIN {X 0,Y 239.802,Z 281.98,A -85,B 0,C 180,E1 -19691.635,E2 -19691.635} C_VEL
LIN {X 0,Y 238.697,Z 287.664,A -85,B 0,C 180,E1 -19692.876,E2 -19692.876} C_VEL
LIN {X 0,Y 237.391,Z 294.012,A -85,B 0,C 180,E1 -19694.547,E2 -19694.547} C_VEL
LIN {X 0,Y 236.236,Z 299.288,A -85,B 0,C 180,E1 -19696.231,E2 -19696.231} C_VEL
LIN {X 0,Y 235.258,Z 303.692,A -85,B 0,C 180,E1 -19697.929,E2 -19697.929} C_VEL
LIN {X 0,Y 234.199,Z 308.869,A -85,B 0,C 180,E1 -19700.5,E2 -19700.5} C_VEL
LIN {X 0,Y 233.612,Z 311.526,A -85,B 0,C 180,E1 -19702.219,E2 -19702.219} C_VEL
LIN {X 0,Y 233.084,Z 314.433,A -85,B 0,C 180,E1 -19704.81,E2 -19704.81} C_VEL
LIN {X 0,Y 232.877,Z 315.701,A -85,B 0,C 180,E1 -19706.539,E2 -19706.539} C_VEL
LIN {X 0,Y 232.762,Z 316.501,A -85,B 0,C 180,E1 -19708.269,E2 -19708.269} C_VEL
LIN {X 0,Y 232.752,Z 316.805,A -85,B 0,C 180,E1 -19710,E2 -19710} C_VEL
LIN {X 0,Y 232.761,Z 316.526,A -85,B 0,C 180,E1 -19711.73,E2 -19711.73} C_VEL
LIN {X 0,Y 232.874,Z 315.777,A -85,B 0,C 180,E1 -19713.46,E2 -19713.46} C_VEL
LIN {X 0,Y 233.225,Z 313.756,A -85,B 0,C 180,E1 -19716.053,E2 -19716.053} C_VEL
LIN {X 0,Y 233.85,Z 310.552,A -85,B 0,C 180,E1 -19718.642,E2 -19718.642} C_VEL
LIN {X 0,Y 234.816,Z 305.896,A -85,B 0,C 180,E1 -19721.218,E2 -19721.218} C_VEL
LIN {X 0,Y 235.919,Z 300.826,A -85,B 0,C 180,E1 -19723.348,E2 -19723.348} C_VEL
LIN {X 0,Y 237.014,Z 295.869,A -85,B 0,C 180,E1 -19725.037,E2 -19725.037} C_VEL
LIN {X 0,Y 238.299,Z 289.886,A -85,B 0,C 180,E1 -19726.711,E2 -19726.711} C_VEL
LIN {X 0,Y 239.718,Z 282.604,A -85,B 0,C 180,E1 -19728.37,E2 -19728.37} C_VEL
LIN {X 0,Y 241.183,Z 274.817,A -85,B 0,C 180,E1 -19729.8,E2 -19729.8} C_VEL
LIN {X 0,Y 242.486,Z 266.601,A -85,B 0,C 180,E1 -19731.018,E2 -19731.018} C_VEL
LIN {X 0,Y 243.926,Z 256.451,A -85,B 0,C 180,E1 -19732.183,E2 -19732.183} C_VEL
LIN {X 0,Y 245.006,Z 244.72,A -85,B 0,C 180,E1 -19733.138,E2 -19733.138} C_VEL
LIN {X 0,Y 245.636,Z 235.107,A -85,B 0,C 180,E1 -19733.65,E2 -19733.65} C_VEL
LIN {X 0,Y 246.159,Z 215.561,A -85,B 0,C 180,E1 -19734.272,E2 -19734.272} C_VEL
LIN {X 0,Y 246.745,Z 192.199,A -85,B 0,C 180,E1 -19734.944,E2 -19734.944} C_VEL
LIN {X 0,Y 244.454,Z 179.716,A -85,B 0,C 180,E1 -19735.593,E2 -19735.593} C_VEL
LIN {X 0,Y 239.136,Z 165.7,A -85,B 0,C 180,E1 -19736.669,E2 -19736.669} C_VEL
LIN {X 0,Y 235.909,Z 158.062,A -85,B 0,C 180,E1 -19737.366,E2 -19737.366} C_VEL
LIN {X 0,Y 235.708,Z 157.189,A -85,B 0,C 180,E1 -19737.622,E2 -19737.622} C_VEL
LIN {X 0,Y 235.023,Z 154.127,A -85,B 0,C 180,E1 -19739.292,E2 -19739.292} C_VEL
LIN {X 0,Y 234.95,Z 154.023,A -85,B 0,C 180,E1 -19743.117,E2 -19743.117} C_VEL
LIN {X 0,Y 234.941,Z 154.019,A -85,B 0,C 180,E1 -19746.746,E2 -19746.746} C_VEL
LIN {X 0,Y 234.942,Z 154.032,A -85,B 0,C 180,E1 -19748.944,E2 -19748.944} C_VEL
LIN {X 0,Y 234.879,Z 154.006,A -85,B 0,C 180,E1 -19753.487,E2 -19753.487} C_VEL
LIN {X 0,Y 234.885,Z 154.039,A -85,B 0,C 180,E1 -19756.513,E2 -19756.513} C_VEL
LIN {X 0,Y 234.917,Z 154.027,A -85,B 0,C 180,E1 -19761.078,E2 -19761.078} C_VEL
LIN {X 0,Y 234.93,Z 154.022,A -85,B 0,C 180,E1 -19765.362,E2 -19765.362} C_VEL
LIN {X 0,Y 234.931,Z 154.034,A -85,B 0,C 180,E1 -19769.432,E2 -19769.432} C_VEL
LIN {X 0,Y 234.993,Z 154.008,A -85,B 0,C 180,E1 -19773.793,E2 -19773.793} C_VEL
LIN {X 0,Y 235.011,Z 154.019,A -85,B 0,C 180,E1 -19778.97,E2 -19778.97} C_VEL
LIN {X 0,Y 235.095,Z 153.998,A -85,B 0,C 180,E1 -19783.059,E2 -19783.059} C_VEL
LIN {X 0,Y 235.146,Z 154.005,A -85,B 0,C 180,E1 -19787.923,E2 -19787.923} C_VEL
LIN {X 0,Y 235.376,Z 153.955,A -85,B 0,C 180,E1 -19791.414,E2 -19791.414} C_VEL
LIN {X 0,Y 235.403,Z 153.966,A -85,B 0,C 180,E1 -19793.141,E2 -19793.141} C_VEL
LIN {X 0,Y 235.595,Z 153.942,A -85,B 0,C 180,E1 -19798.29,E2 -19798.29} C_VEL
LIN {X 0,Y 235.595,Z 153.929,A -85,B 0,C 180,E1 -19801.709,E2 -19801.709} C_VEL
LIN {X 0,Y 235.404,Z 153.972,A -85,B 0,C 180,E1 -19806.858,E2 -19806.858} C_VEL
LIN {X 0,Y 235.237,Z 153.972,A -85,B 0,C 180,E1 -19810.326,E2 -19810.326} C_VEL
LIN {X 0,Y 235.112,Z 154.011,A -85,B 0,C 180,E1 -19815.606,E2 -19815.606} C_VEL
LIN {X 0,Y 235.007,Z 154.006,A -85,B 0,C 180,E1 -19819.205,E2 -19819.205} C_VEL
LIN {X 0,Y 234.948,Z 154.028,A -85,B 0,C 180,E1 -19823.174,E2 -19823.174} C_VEL
LIN {X 0,Y 234.968,Z 154.016,A -85,B 0,C 180,E1 -19826.657,E2 -19826.657} C_VEL
LIN {X 0,Y 234.928,Z 154.032,A -85,B 0,C 180,E1 -19830.6,E2 -19830.6} C_VEL
LIN {X 0,Y 234.217,Z 154.122,A -85,B 0,C 180,E1 -19832.03,E2 -19832.03} C_VEL
LIN {X 0,Y 231.374,Z 154.477,A -85,B 0,C 180,E1 -19834.364,E2 -19834.364} C_VEL
LIN {X 0,Y 228.975,Z 154.782,A -85,B 0,C 180,E1 -19836.267,E2 -19836.267} C_VEL
LIN {X 0,Y 227.931,Z 154.909,A -85,B 0,C 180,E1 -19837.742,E2 -19837.742} C_VEL
LIN {X 0,Y 227.836,Z 154.917,A -85,B 0,C 180,E1 -19838.243,E2 -19838.243} C_VEL
LIN {X 0,Y 227.803,Z 154.877,A -85,B 0,C 180,E1 -19842.744,E2 -19842.744} C_VEL
LIN {X 0,Y 227.804,Z 154.92,A -85,B 0,C 180,E1 -19847.257,E2 -19847.257} C_VEL
LIN {X 0,Y 227.843,Z 154.891,A -85,B 0,C 180,E1 -19851.909,E2 -19851.909} C_VEL
LIN {X 0,Y 227.899,Z 154.91,A -85,B 0,C 180,E1 -19856.534,E2 -19856.534} C_VEL
LIN {X 0,Y 228.143,Z 156.13,A -85,B 0,C 180,E1 -19857.379,E2 -19857.379} C_VEL
LIN {X 0,Y 229.978,Z 164.4,A -85,B 0,C 180,E1 -19861.625,E2 -19861.625} C_VEL
LIN {X 0,Y 230.2,Z 165.453,A -85,B 0,C 180,E1 -19861.941,E2 -19861.941} C_VEL
LIN {X 0,Y 235.317,Z 178.426,A -85,B 0,C 180,E1 -19863.079,E2 -19863.079} C_VEL
LIN {X 0,Y 237.48,Z 190.423,A -85,B 0,C 180,E1 -19863.739,E2 -19863.739} C_VEL
LIN {X 0,Y 239.985,Z 208.087,A -85,B 0,C 180,E1 -19864.606,E2 -19864.606} C_VEL
LIN {X 0,Y 238.934,Z 242.003,A -85,B 0,C 180,E1 -19865.64,E2 -19865.64} C_VEL
LIN {X 0,Y 238.244,Z 251.587,A -85,B 0,C 180,E1 -19866.131,E2 -19866.131} C_VEL
LIN {X 0,Y 237.105,Z 262.549,A -85,B 0,C 180,E1 -19866.973,E2 -19866.973} C_VEL
LIN {X 0,Y 235.636,Z 272.853,A -85,B 0,C 180,E1 -19868.111,E2 -19868.111} C_VEL
LIN {X 0,Y 234.241,Z 281.414,A -85,B 0,C 180,E1 -19869.358,E2 -19869.358} C_VEL
LIN {X 0,Y 232.669,Z 289.471,A -85,B 0,C 180,E1 -19870.823,E2 -19870.823} C_VEL
LIN {X 0,Y 231.27,Z 296.127,A -85,B 0,C 180,E1 -19872.309,E2 -19872.309} C_VEL
LIN {X 0,Y 229.849,Z 302.446,A -85,B 0,C 180,E1 -19874.027,E2 -19874.027} C_VEL
LIN {X 0,Y 228.723,Z 307.699,A -85,B 0,C 180,E1 -19875.77,E2 -19875.77} C_VEL
LIN {X 0,Y 227.737,Z 312.079,A -85,B 0,C 180,E1 -19877.525,E2 -19877.525} C_VEL
LIN {X 0,Y 226.68,Z 317.247,A -85,B 0,C 180,E1 -19880.182,E2 -19880.182} C_VEL
LIN {X 0,Y 225.958,Z 321.041,A -85,B 0,C 180,E1 -19882.854,E2 -19882.854} C_VEL
LIN {X 0,Y 225.665,Z 323.344,A -85,B 0,C 180,E1 -19885.265,E2 -19885.265} C_VEL
LIN {X 0,Y 225.584,Z 324.806,A -85,B 0,C 180,E1 -19888.215,E2 -19888.215} C_VEL
LIN {X 0,Y 225.642,Z 325.099,A -85,B 0,C 180,E1 -19890,E2 -19890} C_VEL
LIN {X 0,Y 225.584,Z 324.797,A -85,B 0,C 180,E1 -19891.786,E2 -19891.786} C_VEL
LIN {X 0,Y 225.664,Z 323.308,A -85,B 0,C 180,E1 -19894.731,E2 -19894.731} C_VEL
LIN {X 0,Y 226.001,Z 320.98,A -85,B 0,C 180,E1 -19897.146,E2 -19897.146} C_VEL
LIN {X 0,Y 226.625,Z 317.165,A -85,B 0,C 180,E1 -19899.821,E2 -19899.821} C_VEL
LIN {X 0,Y 227.733,Z 311.974,A -85,B 0,C 180,E1 -19902.476,E2 -19902.476} C_VEL
LIN {X 0,Y 229.265,Z 305.129,A -85,B 0,C 180,E1 -19905.104,E2 -19905.104} C_VEL
LIN {X 0,Y 230.898,Z 297.653,A -85,B 0,C 180,E1 -19907.264,E2 -19907.264} C_VEL
LIN {X 0,Y 232.467,Z 290.28,A -85,B 0,C 180,E1 -19908.966,E2 -19908.966} C_VEL
LIN {X 0,Y 234.014,Z 282.382,A -85,B 0,C 180,E1 -19910.434,E2 -19910.434} C_VEL
LIN {X 0,Y 235.425,Z 274.032,A -85,B 0,C 180,E1 -19911.68,E2 -19911.68} C_VEL
LIN {X 0,Y 236.889,Z 263.616,A -85,B 0,C 180,E1 -19912.887,E2 -19912.887} C_VEL
LIN {X 0,Y 238.137,Z 251.915,A -85,B 0,C 180,E1 -19913.809,E2 -19913.809} C_VEL
LIN {X 0,Y 238.892,Z 242.942,A -85,B 0,C 180,E1 -19914.273,E2 -19914.273} C_VEL
LIN {X 0,Y 239.812,Z 213.151,A -85,B 0,C 180,E1 -19915.199,E2 -19915.199} C_VEL
LIN {X 0,Y 239.689,Z 206.071,A -85,B 0,C 180,E1 -19915.443,E2 -19915.443} C_VEL
LIN {X 0,Y 235.833,Z 180.715,A -85,B 0,C 180,E1 -19916.729,E2 -19916.729} C_VEL
LIN {X 0,Y 234.3,Z 175.769,A -85,B 0,C 180,E1 -19917.083,E2 -19917.083} C_VEL
LIN {X 0,Y 230.138,Z 165.189,A -85,B 0,C 180,E1 -19918.04,E2 -19918.04} C_VEL
LIN {X 0,Y 228.917,Z 159.627,A -85,B 0,C 180,E1 -19920.725,E2 -19920.725} C_VEL
LIN {X 0,Y 227.911,Z 154.924,A -85,B 0,C 180,E1 -19923.325,E2 -19923.325} C_VEL
LIN {X 0,Y 227.894,Z 154.894,A -85,B 0,C 180,E1 -19926.697,E2 -19926.697} C_VEL
LIN {X 0,Y 227.825,Z 154.91,A -85,B 0,C 180,E1 -19930.377,E2 -19930.377} C_VEL
LIN {X 0,Y 227.826,Z 154.88,A -85,B 0,C 180,E1 -19935.195,E2 -19935.195} C_VEL
LIN {X 0,Y 227.825,Z 154.906,A -85,B 0,C 180,E1 -19939.623,E2 -19939.623} C_VEL
LIN {X 0,Y 227.882,Z 154.903,A -85,B 0,C 180,E1 -19944.129,E2 -19944.129} C_VEL
LIN {X 0,Y 227.872,Z 154.912,A -85,B 0,C 180,E1 -19948.378,E2 -19948.378} C_VEL
LIN {X 0,Y 227.888,Z 154.892,A -85,B 0,C 180,E1 -19952.445,E2 -19952.445} C_VEL
LIN {X 0,Y 227.916,Z 154.907,A -85,B 0,C 180,E1 -19956.368,E2 -19956.368} C_VEL
LIN {X 0,Y 227.944,Z 154.884,A -85,B 0,C 180,E1 -19960.175,E2 -19960.175} C_VEL
LIN {X 0,Y 228.06,Z 154.887,A -85,B 0,C 180,E1 -19963.898,E2 -19963.898} C_VEL
LIN {X 0,Y 228.075,Z 154.878,A -85,B 0,C 180,E1 -19967.544,E2 -19967.544} C_VEL
LIN {X 0,Y 228.269,Z 154.85,A -85,B 0,C 180,E1 -19971.145,E2 -19971.145} C_VEL
LIN {X 0,Y 228.341,Z 154.853,A -85,B 0,C 180,E1 -19972.928,E2 -19972.928} C_VEL
LIN {X 0,Y 228.556,Z 154.805,A -85,B 0,C 180,E1 -19978.238,E2 -19978.238} C_VEL
LIN {X 0,Y 228.556,Z 154.818,A -85,B 0,C 180,E1 -19981.762,E2 -19981.762} C_VEL
LIN {X 0,Y 228.358,Z 154.841,A -85,B 0,C 180,E1 -19987.072,E2 -19987.072} C_VEL
LIN {X 0,Y 228.166,Z 154.864,A -85,B 0,C 180,E1 -19990.65,E2 -19990.65} C_VEL
LIN {X 0,Y 228.068,Z 154.887,A -85,B 0,C 180,E1 -19994.272,E2 -19994.272} C_VEL
LIN {X 0,Y 228.006,Z 154.873,A -85,B 0,C 180,E1 -19997.953,E2 -19997.953} C_VEL
LIN {X 0,Y 227.933,Z 154.903,A -85,B 0,C 180,E1 -20002.329,E2 -20002.329} C_VEL
LIN {X 0,Y 227.945,Z 154.885,A -85,B 0,C 180,E1 -20006.603,E2 -20006.603} C_VEL
LIN {X 0,Y 227.911,Z 154.907,A -85,B 0,C 180,E1 -20010.296,E2 -20010.296} C_VEL
LIN {X 0,Y 227.879,Z 154.896,A -85,B 0,C 180,E1 -20013.72,E2 -20013.72} C_VEL
LIN {X 0,Y 227.846,Z 154.916,A -85,B 0,C 180,E1 -20018.091,E2 -20018.091} C_VEL
LIN {X 0,Y 227.812,Z 154.923,A -85,B 0,C 180,E1 -20022.742,E2 -20022.742} C_VEL
LIN {X 0,Y 227.811,Z 154.884,A -85,B 0,C 180,E1 -20027.257,E2 -20027.257} C_VEL
LIN {X 0,Y 227.872,Z 154.914,A -85,B 0,C 180,E1 -20031.914,E2 -20031.914} C_VEL
LIN {X 0,Y 227.891,Z 154.891,A -85,B 0,C 180,E1 -20036.374,E2 -20036.374} C_VEL
LIN {X 0,Y 227.972,Z 155.113,A -85,B 0,C 180,E1 -20040.354,E2 -20040.354} C_VEL
LIN {X 0,Y 228.613,Z 157.933,A -85,B 0,C 180,E1 -20041.782,E2 -20041.782} C_VEL
LIN {X 0,Y 230.203,Z 161.617,A -85,B 0,C 180,E1 -20042.209,E2 -20042.209} C_VEL
LIN {X 0,Y 236.676,Z 177.457,A -85,B 0,C 180,E1 -20043.565,E2 -20043.565} C_VEL
LIN {X 0,Y 238.706,Z 183.775,A -85,B 0,C 180,E1 -20044.016,E2 -20044.016} C_VEL
LIN {X 0,Y 240.395,Z 193.906,A -85,B 0,C 180,E1 -20044.542,E2 -20044.542} C_VEL
LIN {X 0,Y 239.067,Z 234.213,A -85,B 0,C 180,E1 -20045.753,E2 -20045.753} C_VEL
LIN {X 0,Y 238.429,Z 244.183,A -85,B 0,C 180,E1 -20046.278,E2 -20046.278} C_VEL
LIN {X 0,Y 237.385,Z 255.455,A -85,B 0,C 180,E1 -20047.18,E2 -20047.18} C_VEL
LIN {X 0,Y 235.927,Z 265.812,A -85,B 0,C 180,E1 -20048.368,E2 -20048.368} C_VEL
LIN {X 0,Y 234.6,Z 274.194,A -85,B 0,C 180,E1 -20049.619,E2 -20049.619} C_VEL
LIN {X 0,Y 233.065,Z 282.112,A -85,B 0,C 180,E1 -20051.085,E2 -20051.085} C_VEL
LIN {X 0,Y 231.919,Z 287.796,A -85,B 0,C 180,E1 -20052.36,E2 -20052.36} C_VEL
LIN {X 0,Y 230.567,Z 294.142,A -85,B 0,C 180,E1 -20054.077,E2 -20054.077} C_VEL
LIN {X 0,Y 229.346,Z 299.418,A -85,B 0,C 180,E1 -20055.809,E2 -20055.809} C_VEL
LIN {X 0,Y 228.306,Z 303.822,A -85,B 0,C 180,E1 -20057.556,E2 -20057.556} C_VEL
LIN {X 0,Y 227.183,Z 308.999,A -85,B 0,C 180,E1 -20060.203,E2 -20060.203} C_VEL
LIN {X 0,Y 226.58,Z 311.655,A -85,B 0,C 180,E1 -20061.976,E2 -20061.976} C_VEL
LIN {X 0,Y 226.011,Z 314.562,A -85,B 0,C 180,E1 -20064.647,E2 -20064.647} C_VEL
LIN {X 0,Y 225.792,Z 315.83,A -85,B 0,C 180,E1 -20066.43,E2 -20066.43} C_VEL
LIN {X 0,Y 225.664,Z 316.629,A -85,B 0,C 180,E1 -20068.215,E2 -20068.215} C_VEL
LIN {X 0,Y 225.668,Z 316.933,A -85,B 0,C 180,E1 -20070,E2 -20070} C_VEL
LIN {X 0,Y 225.663,Z 316.654,A -85,B 0,C 180,E1 -20071.784,E2 -20071.784} C_VEL
LIN {X 0,Y 225.787,Z 315.905,A -85,B 0,C 180,E1 -20073.569,E2 -20073.569} C_VEL
LIN {X 0,Y 226.108,Z 314.164,A -85,B 0,C 180,E1 -20075.932,E2 -20075.932} C_VEL
LIN {X 0,Y 226.571,Z 311.832,A -85,B 0,C 180,E1 -20078.023,E2 -20078.023} C_VEL
LIN {X 0,Y 227.145,Z 309.232,A -85,B 0,C 180,E1 -20079.797,E2 -20079.797} C_VEL
LIN {X 0,Y 228.271,Z 304.118,A -85,B 0,C 180,E1 -20082.445,E2 -20082.445} C_VEL
LIN {X 0,Y 229.604,Z 298.613,A -85,B 0,C 180,E1 -20084.627,E2 -20084.627} C_VEL
LIN {X 0,Y 231.18,Z 291.693,A -85,B 0,C 180,E1 -20086.786,E2 -20086.786} C_VEL
LIN {X 0,Y 232.79,Z 283.748,A -85,B 0,C 180,E1 -20088.709,E2 -20088.709} C_VEL
LIN {X 0,Y 234.282,Z 276.169,A -85,B 0,C 180,E1 -20090.18,E2 -20090.18} C_VEL
LIN {X 0,Y 235.685,Z 268.223,A -85,B 0,C 180,E1 -20091.425,E2 -20091.425} C_VEL
LIN {X 0,Y 236.909,Z 260.01,A -85,B 0,C 180,E1 -20092.453,E2 -20092.453} C_VEL
LIN {X 0,Y 237.922,Z 251.478,A -85,B 0,C 180,E1 -20093.29,E2 -20093.29} C_VEL
LIN {X 0,Y 238.713,Z 241.853,A -85,B 0,C 180,E1 -20093.993,E2 -20093.993} C_VEL
LIN {X 0,Y 239.228,Z 232.017,A -85,B 0,C 180,E1 -20094.467,E2 -20094.467} C_VEL
LIN {X 0,Y 240.357,Z 193.399,A -85,B 0,C 180,E1 -20095.619,E2 -20095.619} C_VEL
LIN {X 0,Y 238.22,Z 181.656,A -85,B 0,C 180,E1 -20096.253,E2 -20096.253} C_VEL
LIN {X 0,Y 231.729,Z 165.031,A -85,B 0,C 180,E1 -20097.619,E2 -20097.619} C_VEL
LIN {X 0,Y 228.681,Z 158.151,A -85,B 0,C 180,E1 -20098.317,E2 -20098.317} C_VEL
LIN {X 0,Y 228.367,Z 156.8,A -85,B 0,C 180,E1 -20098.853,E2 -20098.853} C_VEL
LIN {X 0,Y 227.947,Z 154.999,A -85,B 0,C 180,E1 -20099.923,E2 -20099.923} C_VEL
LIN {X 0,Y 227.89,Z 154.892,A -85,B 0,C 180,E1 -20103.718,E2 -20103.718} C_VEL
LIN {X 0,Y 227.87,Z 154.913,A -85,B 0,C 180,E1 -20108.085,E2 -20108.085} C_VEL
LIN {X 0,Y 227.808,Z 154.881,A -85,B 0,C 180,E1 -20112.742,E2 -20112.742} C_VEL
LIN {X 0,Y 227.809,Z 154.922,A -85,B 0,C 180,E1 -20117.257,E2 -20117.257} C_VEL
LIN {X 0,Y 227.843,Z 154.915,A -85,B 0,C 180,E1 -20121.908,E2 -20121.908} C_VEL
LIN {X 0,Y 227.879,Z 154.896,A -85,B 0,C 180,E1 -20126.377,E2 -20126.377} C_VEL
LIN {X 0,Y 227.918,Z 154.906,A -85,B 0,C 180,E1 -20130.437,E2 -20130.437} C_VEL
LIN {X 0,Y 227.928,Z 154.89,A -85,B 0,C 180,E1 -20134.426,E2 -20134.426} C_VEL
LIN {X 0,Y 227.961,Z 154.901,A -85,B 0,C 180,E1 -20138.287,E2 -20138.287} C_VEL
LIN {X 0,Y 228.034,Z 154.874,A -85,B 0,C 180,E1 -20142.826,E2 -20142.826} C_VEL
LIN {X 0,Y 228.094,Z 154.883,A -85,B 0,C 180,E1 -20147.544,E2 -20147.544} C_VEL
LIN {X 0,Y 228.305,Z 154.834,A -85,B 0,C 180,E1 -20151.146,E2 -20151.146} C_VEL
LIN {X 0,Y 228.354,Z 154.84,A -85,B 0,C 180,E1 -20152.928,E2 -20152.928} C_VEL
LIN {X 0,Y 228.554,Z 154.819,A -85,B 0,C 180,E1 -20158.238,E2 -20158.238} C_VEL
LIN {X 0,Y 228.554,Z 154.805,A -85,B 0,C 180,E1 -20161.762,E2 -20161.762} C_VEL
LIN {X 0,Y 228.355,Z 154.851,A -85,B 0,C 180,E1 -20167.071,E2 -20167.071} C_VEL
LIN {X 0,Y 228.162,Z 154.852,A -85,B 0,C 180,E1 -20170.65,E2 -20170.65} C_VEL
LIN {X 0,Y 228.064,Z 154.887,A -85,B 0,C 180,E1 -20174.272,E2 -20174.272} C_VEL
LIN {X 0,Y 228.002,Z 154.885,A -85,B 0,C 180,E1 -20177.953,E2 -20177.953} C_VEL
LIN {X 0,Y 227.929,Z 154.902,A -85,B 0,C 180,E1 -20182.329,E2 -20182.329} C_VEL
LIN {X 0,Y 227.942,Z 154.891,A -85,B 0,C 180,E1 -20186.603,E2 -20186.603} C_VEL
LIN {X 0,Y 227.889,Z 154.907,A -85,B 0,C 180,E1 -20190.575,E2 -20190.575} C_VEL
LIN {X 0,Y 227.876,Z 154.904,A -85,B 0,C 180,E1 -20193.72,E2 -20193.72} C_VEL
LIN {X 0,Y 227.842,Z 154.918,A -85,B 0,C 180,E1 -20198.091,E2 -20198.091} C_VEL
LIN {X 0,Y 227.836,Z 154.917,A -85,B 0,C 180,E1 -20198.243,E2 -20198.243} C_VEL
LIN {X 0,Y 227.141,Z 154.997,A -85,B 0,C 180,E1 -20199.718,E2 -20199.718} C_VEL
LIN {X 0,Y 224.286,Z 155.327,A -85,B 0,C 180,E1 -20202.126,E2 -20202.126} C_VEL
LIN {X 0,Y 221.871,Z 155.623,A -85,B 0,C 180,E1 -20204.09,E2 -20204.09} C_VEL
LIN {X 0,Y 220.832,Z 155.763,A -85,B 0,C 180,E1 -20205.615,E2 -20205.615} C_VEL
LIN {X 0,Y 220.745,Z 155.78,A -85,B 0,C 180,E1 -20206.132,E2 -20206.132} C_VEL
LIN {X 0,Y 220.805,Z 155.772,A -85,B 0,C 180,E1 -20210.463,E2 -20210.463} C_VEL
LIN {X 0,Y 220.801,Z 155.791,A -85,B 0,C 180,E1 -20215.046,E2 -20215.046} C_VEL
LIN {X 0,Y 220.868,Z 156.003,A -85,B 0,C 180,E1 -20216.152,E2 -20216.152} C_VEL
LIN {X 0,Y 222.85,Z 164.792,A -85,B 0,C 180,E1 -20220.845,E2 -20220.845} C_VEL
LIN {X 0,Y 224.215,Z 168.27,A -85,B 0,C 180,E1 -20221.273,E2 -20221.273} C_VEL
LIN {X 0,Y 229.416,Z 181.391,A -85,B 0,C 180,E1 -20222.434,E2 -20222.434} C_VEL
LIN {X 0,Y 232.958,Z 204.056,A -85,B 0,C 180,E1 -20223.651,E2 -20223.651} C_VEL
LIN {X 0,Y 233.563,Z 210.06,A -85,B 0,C 180,E1 -20223.926,E2 -20223.926} C_VEL
LIN {X 0,Y 232.439,Z 242.841,A -85,B 0,C 180,E1 -20224.957,E2 -20224.957} C_VEL
LIN {X 0,Y 231.555,Z 254.005,A -85,B 0,C 180,E1 -20225.579,E2 -20225.579} C_VEL
LIN {X 0,Y 230.159,Z 265.56,A -85,B 0,C 180,E1 -20226.612,E2 -20226.612} C_VEL
LIN {X 0,Y 228.808,Z 274.231,A -85,B 0,C 180,E1 -20227.66,E2 -20227.66} C_VEL
LIN {X 0,Y 227.399,Z 282.521,A -85,B 0,C 180,E1 -20228.944,E2 -20228.944} C_VEL
LIN {X 0,Y 225.758,Z 290.367,A -85,B 0,C 180,E1 -20230.449,E2 -20230.449} C_VEL
LIN {X 0,Y 224.131,Z 297.708,A -85,B 0,C 180,E1 -20232.199,E2 -20232.199} C_VEL
LIN {X 0,Y 222.398,Z 305.154,A -85,B 0,C 180,E1 -20234.419,E2 -20234.419} C_VEL
LIN {X 0,Y 220.792,Z 311.952,A -85,B 0,C 180,E1 -20237.126,E2 -20237.126} C_VEL
LIN {X 0,Y 219.662,Z 317.119,A -85,B 0,C 180,E1 -20239.865,E2 -20239.865} C_VEL
LIN {X 0,Y 218.922,Z 320.914,A -85,B 0,C 180,E1 -20242.623,E2 -20242.623} C_VEL
LIN {X 0,Y 218.574,Z 323.412,A -85,B 0,C 180,E1 -20245.391,E2 -20245.391} C_VEL
LIN {X 0,Y 218.488,Z 324.678,A -85,B 0,C 180,E1 -20248.157,E2 -20248.157} C_VEL
LIN {X 0,Y 218.541,Z 324.971,A -85,B 0,C 180,E1 -20250,E2 -20250} C_VEL
LIN {X 0,Y 218.488,Z 324.669,A -85,B 0,C 180,E1 -20251.844,E2 -20251.844} C_VEL
LIN {X 0,Y 218.55,Z 323.429,A -85,B 0,C 180,E1 -20254.531,E2 -20254.531} C_VEL
LIN {X 0,Y 218.947,Z 320.85,A -85,B 0,C 180,E1 -20257.377,E2 -20257.377} C_VEL
LIN {X 0,Y 219.62,Z 317.035,A -85,B 0,C 180,E1 -20260.138,E2 -20260.138} C_VEL
LIN {X 0,Y 220.788,Z 311.844,A -85,B 0,C 180,E1 -20262.875,E2 -20262.875} C_VEL
LIN {X 0,Y 222.384,Z 304.998,A -85,B 0,C 180,E1 -20265.583,E2 -20265.583} C_VEL
LIN {X 0,Y 224.129,Z 297.522,A -85,B 0,C 180,E1 -20267.802,E2 -20267.802} C_VEL
LIN {X 0,Y 225.768,Z 290.148,A -85,B 0,C 180,E1 -20269.551,E2 -20269.551} C_VEL
LIN {X 0,Y 227.369,Z 282.25,A -85,B 0,C 180,E1 -20271.059,E2 -20271.059} C_VEL
LIN {X 0,Y 228.849,Z 273.899,A -85,B 0,C 180,E1 -20272.337,E2 -20272.337} C_VEL
LIN {X 0,Y 230.436,Z 262.97,A -85,B 0,C 180,E1 -20273.624,E2 -20273.624} C_VEL
LIN {X 0,Y 231.679,Z 251.815,A -85,B 0,C 180,E1 -20274.513,E2 -20274.513} C_VEL
LIN {X 0,Y 232.439,Z 242.801,A -85,B 0,C 180,E1 -20274.992,E2 -20274.992} C_VEL
LIN {X 0,Y 233.338,Z 214.75,A -85,B 0,C 180,E1 -20275.891,E2 -20275.891} C_VEL
LIN {X 0,Y 233.368,Z 207.622,A -85,B 0,C 180,E1 -20276.126,E2 -20276.126} C_VEL
LIN {X 0,Y 229.645,Z 182.605,A -85,B 0,C 180,E1 -20277.439,E2 -20277.439} C_VEL
LIN {X 0,Y 226.967,Z 174.984,A -85,B 0,C 180,E1 -20278.055,E2 -20278.055} C_VEL
LIN {X 0,Y 222.951,Z 165.21,A -85,B 0,C 180,E1 -20278.999,E2 -20278.999} C_VEL
LIN {X 0,Y 222.675,Z 163.969,A -85,B 0,C 180,E1 -20279.454,E2 -20279.454} C_VEL
LIN {X 0,Y 220.83,Z 155.86,A -85,B 0,C 180,E1 -20283.926,E2 -20283.926} C_VEL
LIN {X 0,Y 220.812,Z 155.769,A -85,B 0,C 180,E1 -20287.279,E2 -20287.279} C_VEL
LIN {X 0,Y 220.768,Z 155.799,A -85,B 0,C 180,E1 -20291.954,E2 -20291.954} C_VEL
LIN {X 0,Y 220.768,Z 155.753,A -85,B 0,C 180,E1 -20295.545,E2 -20295.545} C_VEL
LIN {X 0,Y 220.807,Z 155.789,A -85,B 0,C 180,E1 -20300.463,E2 -20300.463} C_VEL
LIN {X 0,Y 220.803,Z 155.78,A -85,B 0,C 180,E1 -20305.046,E2 -20305.046} C_VEL
LIN {X 0,Y 220.87,Z 155.783,A -85,B 0,C 180,E1 -20309.395,E2 -20309.395} C_VEL
LIN {X 0,Y 220.897,Z 155.769,A -85,B 0,C 180,E1 -20313.55,E2 -20313.55} C_VEL
LIN {X 0,Y 220.88,Z 155.779,A -85,B 0,C 180,E1 -20317.554,E2 -20317.554} C_VEL
LIN {X 0,Y 220.986,Z 155.761,A -85,B 0,C 180,E1 -20322.571,E2 -20322.571} C_VEL
LIN {X 0,Y 221.014,Z 155.758,A -85,B 0,C 180,E1 -20327.139,E2 -20327.139} C_VEL
LIN {X 0,Y 221.207,Z 155.724,A -85,B 0,C 180,E1 -20330.86,E2 -20330.86} C_VEL
LIN {X 0,Y 221.274,Z 155.731,A -85,B 0,C 180,E1 -20332.701,E2 -20332.701} C_VEL
LIN {X 0,Y 221.514,Z 155.681,A -85,B 0,C 180,E1 -20338.182,E2 -20338.182} C_VEL
LIN {X 0,Y 221.514,Z 155.696,A -85,B 0,C 180,E1 -20341.818,E2 -20341.818} C_VEL
LIN {X 0,Y 221.292,Z 155.716,A -85,B 0,C 180,E1 -20347.299,E2 -20347.299} C_VEL
LIN {X 0,Y 221.115,Z 155.743,A -85,B 0,C 180,E1 -20350.994,E2 -20350.994} C_VEL
LIN {X 0,Y 221.019,Z 155.753,A -85,B 0,C 180,E1 -20356.63,E2 -20356.63} C_VEL
LIN {X 0,Y 220.895,Z 155.774,A -85,B 0,C 180,E1 -20360.486,E2 -20360.486} C_VEL
LIN {X 0,Y 220.87,Z 155.779,A -85,B 0,C 180,E1 -20364.435,E2 -20364.435} C_VEL
LIN {X 0,Y 220.839,Z 155.781,A -85,B 0,C 180,E1 -20368.513,E2 -20368.513} C_VEL
LIN {X 0,Y 220.82,Z 155.779,A -85,B 0,C 180,E1 -20372.756,E2 -20372.756} C_VEL
LIN {X 0,Y 220.812,Z 155.792,A -85,B 0,C 180,E1 -20377.278,E2 -20377.278} C_VEL
LIN {X 0,Y 220.771,Z 155.796,A -85,B 0,C 180,E1 -20381.952,E2 -20381.952} C_VEL
LIN {X 0,Y 220.772,Z 155.775,A -85,B 0,C 180,E1 -20385.545,E2 -20385.545} C_VEL
LIN {X 0,Y 220.811,Z 155.784,A -85,B 0,C 180,E1 -20390.464,E2 -20390.464} C_VEL
LIN {X 0,Y 220.834,Z 155.783,A -85,B 0,C 180,E1 -20392.794,E2 -20392.794} C_VEL
LIN {X 0,Y 220.825,Z 155.782,A -85,B 0,C 180,E1 -20397.245,E2 -20397.245} C_VEL
LIN {X 0,Y 220.909,Z 156.008,A -85,B 0,C 180,E1 -20399.711,E2 -20399.711} C_VEL
LIN {X 0,Y 221.415,Z 158.167,A -85,B 0,C 180,E1 -20400.794,E2 -20400.794} C_VEL
LIN {X 0,Y 224.326,Z 164.653,A -85,B 0,C 180,E1 -20401.518,E2 -20401.518} C_VEL
LIN {X 0,Y 230.554,Z 179.81,A -85,B 0,C 180,E1 -20402.881,E2 -20402.881} C_VEL
LIN {X 0,Y 232.57,Z 186.129,A -85,B 0,C 180,E1 -20403.352,E2 -20403.352} C_VEL
LIN {X 0,Y 233.986,Z 195.752,A -85,B 0,C 180,E1 -20403.85,E2 -20403.85} C_VEL
LIN {X 0,Y 232.609,Z 234.546,A -85,B 0,C 180,E1 -20405.044,E2 -20405.044} C_VEL
LIN {X 0,Y 231.919,Z 244.937,A -85,B 0,C 180,E1 -20405.614,E2 -20405.614} C_VEL
LIN {X 0,Y 230.637,Z 257.137,A -85,B 0,C 180,E1 -20406.663,E2 -20406.663} C_VEL
LIN {X 0,Y 229.353,Z 265.945,A -85,B 0,C 180,E1 -20407.715,E2 -20407.715} C_VEL
LIN {X 0,Y 227.975,Z 274.327,A -85,B 0,C 180,E1 -20408.999,E2 -20408.999} C_VEL
LIN {X 0,Y 226.372,Z 282.244,A -85,B 0,C 180,E1 -20410.503,E2 -20410.503} C_VEL
LIN {X 0,Y 224.818,Z 289.624,A -85,B 0,C 180,E1 -20412.254,E2 -20412.254} C_VEL
LIN {X 0,Y 223.101,Z 297.1,A -85,B 0,C 180,E1 -20414.468,E2 -20414.468} C_VEL
LIN {X 0,Y 221.382,Z 303.952,A -85,B 0,C 180,E1 -20417.16,E2 -20417.16} C_VEL
LIN {X 0,Y 220.19,Z 309.129,A -85,B 0,C 180,E1 -20419.889,E2 -20419.889} C_VEL
LIN {X 0,Y 219.547,Z 311.785,A -85,B 0,C 180,E1 -20421.717,E2 -20421.717} C_VEL
LIN {X 0,Y 218.955,Z 314.691,A -85,B 0,C 180,E1 -20424.474,E2 -20424.474} C_VEL
LIN {X 0,Y 218.709,Z 315.959,A -85,B 0,C 180,E1 -20426.315,E2 -20426.315} C_VEL
LIN {X 0,Y 218.569,Z 316.758,A -85,B 0,C 180,E1 -20428.157,E2 -20428.157} C_VEL
LIN {X 0,Y 218.586,Z 317.061,A -85,B 0,C 180,E1 -20430,E2 -20430} C_VEL
LIN {X 0,Y 218.568,Z 316.782,A -85,B 0,C 180,E1 -20431.842,E2 -20431.842} C_VEL
LIN {X 0,Y 218.705,Z 316.033,A -85,B 0,C 180,E1 -20433.684,E2 -20433.684} C_VEL
LIN {X 0,Y 218.972,Z 314.616,A -85,B 0,C 180,E1 -20435.753,E2 -20435.753} C_VEL
LIN {X 0,Y 219.539,Z 311.96,A -85,B 0,C 180,E1 -20438.282,E2 -20438.282} C_VEL
LIN {X 0,Y 220.161,Z 309.359,A -85,B 0,C 180,E1 -20440.111,E2 -20440.111} C_VEL
LIN {X 0,Y 221.354,Z 304.245,A -85,B 0,C 180,E1 -20442.841,E2 -20442.841} C_VEL
LIN {X 0,Y 222.731,Z 298.739,A -85,B 0,C 180,E1 -20445.088,E2 -20445.088} C_VEL
LIN {X 0,Y 224.387,Z 291.819,A -85,B 0,C 180,E1 -20447.31,E2 -20447.31} C_VEL
LIN {X 0,Y 226.086,Z 283.873,A -85,B 0,C 180,E1 -20449.285,E2 -20449.285} C_VEL
LIN {X 0,Y 227.647,Z 276.293,A -85,B 0,C 180,E1 -20450.795,E2 -20450.795} C_VEL
LIN {X 0,Y 229.105,Z 268.346,A -85,B 0,C 180,E1 -20452.072,E2 -20452.072} C_VEL
LIN {X 0,Y 230.381,Z 260.132,A -85,B 0,C 180,E1 -20453.126,E2 -20453.126} C_VEL
LIN {X 0,Y 231.372,Z 252.238,A -85,B 0,C 180,E1 -20453.927,E2 -20453.927} C_VEL
LIN {X 0,Y 232.19,Z 243.057,A -85,B 0,C 180,E1 -20454.633,E2 -20454.633} C_VEL
LIN {X 0,Y 232.783,Z 233.883,A -85,B 0,C 180,E1 -20455.11,E2 -20455.11} C_VEL
LIN {X 0,Y 233.904,Z 194.035,A -85,B 0,C 180,E1 -20456.361,E2 -20456.361} C_VEL
LIN {X 0,Y 232.113,Z 184.07,A -85,B 0,C 180,E1 -20456.92,E2 -20456.92} C_VEL
LIN {X 0,Y 225.769,Z 167.868,A -85,B 0,C 180,E1 -20458.317,E2 -20458.317} C_VEL
LIN {X 0,Y 221.484,Z 158.349,A -85,B 0,C 180,E1 -20459.318,E2 -20459.318} C_VEL
LIN {X 0,Y 221.173,Z 157.19,A -85,B 0,C 180,E1 -20459.753,E2 -20459.753} C_VEL
LIN {X 0,Y 220.869,Z 155.873,A -85,B 0,C 180,E1 -20460.604,E2 -20460.604} C_VEL
LIN {X 0,Y 220.815,Z 155.764,A -85,B 0,C 180,E1 -20464.952,E2 -20464.952} C_VEL
LIN {X 0,Y 220.838,Z 155.781,A -85,B 0,C 180,E1 -20467.287,E2 -20467.287} C_VEL
LIN {X 0,Y 220.771,Z 155.758,A -85,B 0,C 180,E1 -20471.952,E2 -20471.952} C_VEL
LIN {X 0,Y 220.77,Z 155.789,A -85,B 0,C 180,E1 -20475.545,E2 -20475.545} C_VEL
LIN {X 0,Y 220.806,Z 155.782,A -85,B 0,C 180,E1 -20480.463,E2 -20480.463} C_VEL
LIN {X 0,Y 220.801,Z 155.783,A -85,B 0,C 180,E1 -20485.045,E2 -20485.045} C_VEL
LIN {X 0,Y 220.867,Z 155.787,A -85,B 0,C 180,E1 -20489.395,E2 -20489.395} C_VEL
LIN {X 0,Y 220.895,Z 155.762,A -85,B 0,C 180,E1 -20493.549,E2 -20493.549} C_VEL
LIN {X 0,Y 220.877,Z 155.783,A -85,B 0,C 180,E1 -20497.553,E2 -20497.553} C_VEL
LIN {X 0,Y 220.983,Z 155.749,A -85,B 0,C 180,E1 -20502.571,E2 -20502.571} C_VEL
LIN {X 0,Y 221.026,Z 155.763,A -85,B 0,C 180,E1 -20507.139,E2 -20507.139} C_VEL
LIN {X 0,Y 221.235,Z 155.714,A -85,B 0,C 180,E1 -20510.86,E2 -20510.86} C_VEL
LIN {X 0,Y 221.289,Z 155.716,A -85,B 0,C 180,E1 -20512.701,E2 -20512.701} C_VEL
LIN {X 0,Y 221.512,Z 155.696,A -85,B 0,C 180,E1 -20518.182,E2 -20518.182} C_VEL
LIN {X 0,Y 221.512,Z 155.682,A -85,B 0,C 180,E1 -20521.818,E2 -20521.818} C_VEL
LIN {X 0,Y 221.306,Z 155.727,A -85,B 0,C 180,E1 -20527.298,E2 -20527.298} C_VEL
LIN {X 0,Y 221.111,Z 155.73,A -85,B 0,C 180,E1 -20530.994,E2 -20530.994} C_VEL
LIN {X 0,Y 221.015,Z 155.765,A -85,B 0,C 180,E1 -20536.63,E2 -20536.63} C_VEL
LIN {X 0,Y 220.891,Z 155.765,A -85,B 0,C 180,E1 -20540.486,E2 -20540.486} C_VEL
LIN {X 0,Y 220.866,Z 155.785,A -85,B 0,C 180,E1 -20544.435,E2 -20544.435} C_VEL
LIN {X 0,Y 220.835,Z 155.773,A -85,B 0,C 180,E1 -20548.513,E2 -20548.513} C_VEL
LIN {X 0,Y 220.816,Z 155.787,A -85,B 0,C 180,E1 -20552.756,E2 -20552.756} C_VEL
LIN {X 0,Y 220.809,Z 155.793,A -85,B 0,C 180,E1 -20557.279,E2 -20557.279} C_VEL
LIN {X 0,Y 220.792,Z 155.781,A -85,B 0,C 180,E1 -20560.188,E2 -20560.188} C_VEL
LIN {X 0,Y 220.765,Z 155.755,A -85,B 0,C 180,E1 -20564.456,E2 -20564.456} C_VEL
LIN {X 0,Y 220.745,Z 155.78,A -85,B 0,C 180,E1 -20566.132,E2 -20566.132} C_VEL
LIN {X 0,Y 220.071,Z 155.886,A -85,B 0,C 180,E1 -20567.656,E2 -20567.656} C_VEL
LIN {X 0,Y 217.235,Z 156.223,A -85,B 0,C 180,E1 -20570.144,E2 -20570.144} C_VEL
LIN {X 0,Y 214.835,Z 156.515,A -85,B 0,C 180,E1 -20572.176,E2 -20572.176} C_VEL
LIN {X 0,Y 213.812,Z 156.652,A -85,B 0,C 180,E1 -20573.753,E2 -20573.753} C_VEL
LIN {X 0,Y 213.732,Z 156.671,A -85,B 0,C 180,E1 -20574.288,E2 -20574.288} C_VEL
LIN {X 0,Y 213.79,Z 156.91,A -85,B 0,C 180,E1 -20575.449,E2 -20575.449} C_VEL
LIN {X 0,Y 215.563,Z 164.66,A -85,B 0,C 180,E1 -20579.764,E2 -20579.764} C_VEL
LIN {X 0,Y 217.168,Z 168.415,A -85,B 0,C 180,E1 -20580.259,E2 -20580.259} C_VEL
LIN {X 0,Y 223.439,Z 183.99,A -85,B 0,C 180,E1 -20581.727,E2 -20581.727} C_VEL
LIN {X 0,Y 227.033,Z 208.164,A -85,B 0,C 180,E1 -20583.055,E2 -20583.055} C_VEL
LIN {X 0,Y 226.938,Z 217.325,A -85,B 0,C 180,E1 -20583.36,E2 -20583.36} C_VEL
LIN {X 0,Y 226.035,Z 242.729,A -85,B 0,C 180,E1 -20584.197,E2 -20584.197} C_VEL
LIN {X 0,Y 225.147,Z 253.438,A -85,B 0,C 180,E1 -20584.802,E2 -20584.802} C_VEL
LIN {X 0,Y 223.656,Z 265.437,A -85,B 0,C 180,E1 -20585.89,E2 -20585.89} C_VEL
LIN {X 0,Y 222.274,Z 274.108,A -85,B 0,C 180,E1 -20586.966,E2 -20586.966} C_VEL
LIN {X 0,Y 220.781,Z 282.396,A -85,B 0,C 180,E1 -20588.282,E2 -20588.282} C_VEL
LIN {X 0,Y 219.085,Z 290.242,A -85,B 0,C 180,E1 -20589.828,E2 -20589.828} C_VEL
LIN {X 0,Y 217.382,Z 297.582,A -85,B 0,C 180,E1 -20591.626,E2 -20591.626} C_VEL
LIN {X 0,Y 215.552,Z 305.028,A -85,B 0,C 180,E1 -20593.911,E2 -20593.911} C_VEL
LIN {X 0,Y 214.124,Z 310.866,A -85,B 0,C 180,E1 -20596.234,E2 -20596.234} C_VEL
LIN {X 0,Y 213.013,Z 315.469,A -85,B 0,C 180,E1 -20598.583,E2 -20598.583} C_VEL
LIN {X 0,Y 212.377,Z 318.463,A -85,B 0,C 180,E1 -20600.477,E2 -20600.477} C_VEL
LIN {X 0,Y 211.874,Z 320.786,A -85,B 0,C 180,E1 -20602.376,E2 -20602.376} C_VEL
LIN {X 0,Y 211.472,Z 323.459,A -85,B 0,C 180,E1 -20605.566,E2 -20605.566} C_VEL
LIN {X 0,Y 211.394,Z 324.549,A -85,B 0,C 180,E1 -20608.095,E2 -20608.095} C_VEL
LIN {X 0,Y 211.442,Z 324.842,A -85,B 0,C 180,E1 -20610,E2 -20610} C_VEL
LIN {X 0,Y 211.394,Z 324.54,A -85,B 0,C 180,E1 -20611.906,E2 -20611.906} C_VEL
LIN {X 0,Y 211.472,Z 323.431,A -85,B 0,C 180,E1 -20614.435,E2 -20614.435} C_VEL
LIN {X 0,Y 211.888,Z 320.721,A -85,B 0,C 180,E1 -20617.625,E2 -20617.625} C_VEL
LIN {X 0,Y 212.313,Z 318.389,A -85,B 0,C 180,E1 -20619.527,E2 -20619.527} C_VEL
LIN {X 0,Y 213.385,Z 313.632,A -85,B 0,C 180,E1 -20622.362,E2 -20622.362} C_VEL
LIN {X 0,Y 214.684,Z 308.484,A -85,B 0,C 180,E1 -20624.697,E2 -20624.697} C_VEL
LIN {X 0,Y 215.873,Z 303.45,A -85,B 0,C 180,E1 -20626.551,E2 -20626.551} C_VEL
LIN {X 0,Y 217.385,Z 297.391,A -85,B 0,C 180,E1 -20628.374,E2 -20628.374} C_VEL
LIN {X 0,Y 219.091,Z 290.017,A -85,B 0,C 180,E1 -20630.172,E2 -20630.172} C_VEL
LIN {X 0,Y 220.75,Z 282.117,A -85,B 0,C 180,E1 -20631.722,E2 -20631.722} C_VEL
LIN {X 0,Y 222.302,Z 273.766,A -85,B 0,C 180,E1 -20633.032,E2 -20633.032} C_VEL
LIN {X 0,Y 223.873,Z 263.347,A -85,B 0,C 180,E1 -20634.301,E2 -20634.301} C_VEL
LIN {X 0,Y 225.242,Z 251.779,A -85,B 0,C 180,E1 -20635.254,E2 -20635.254} C_VEL
LIN {X 0,Y 226.026,Z 242.773,A -85,B 0,C 180,E1 -20635.747,E2 -20635.747} C_VEL
LIN {X 0,Y 226.882,Z 217.216,A -85,B 0,C 180,E1 -20636.594,E2 -20636.594} C_VEL
LIN {X 0,Y 227.011,Z 208.708,A -85,B 0,C 180,E1 -20636.873,E2 -20636.873} C_VEL
LIN {X 0,Y 223.348,Z 183.893,A -85,B 0,C 180,E1 -20638.229,E2 -20638.229} C_VEL
LIN {X 0,Y 218.283,Z 171.147,A -85,B 0,C 180,E1 -20639.411,E2 -20639.411} C_VEL
LIN {X 0,Y 215.614,Z 164.928,A -85,B 0,C 180,E1 -20640.105,E2 -20640.105} C_VEL
LIN {X 0,Y 214.872,Z 161.669,A -85,B 0,C 180,E1 -20641.745,E2 -20641.745} C_VEL
LIN {X 0,Y 213.77,Z 156.688,A -85,B 0,C 180,E1 -20644.724,E2 -20644.724} C_VEL
LIN {X 0,Y 213.723,Z 156.648,A -85,B 0,C 180,E1 -20648.667,E2 -20648.667} C_VEL
LIN {X 0,Y 213.711,Z 156.675,A -85,B 0,C 180,E1 -20651.126,E2 -20651.126} C_VEL
LIN {X 0,Y 213.704,Z 156.661,A -85,B 0,C 180,E1 -20653.68,E2 -20653.68} C_VEL
LIN {X 0,Y 213.703,Z 156.627,A -85,B 0,C 180,E1 -20656.345,E2 -20656.345} C_VEL
LIN {X 0,Y 213.717,Z 156.653,A -85,B 0,C 180,E1 -20659.144,E2 -20659.144} C_VEL
LIN {X 0,Y 213.745,Z 156.665,A -85,B 0,C 180,E1 -20663.712,E2 -20663.712} C_VEL
LIN {X 0,Y 213.797,Z 156.667,A -85,B 0,C 180,E1 -20668.725,E2 -20668.725} C_VEL
LIN {X 0,Y 213.828,Z 156.642,A -85,B 0,C 180,E1 -20672.604,E2 -20672.604} C_VEL
LIN {X 0,Y 213.854,Z 156.658,A -85,B 0,C 180,E1 -20676.953,E2 -20676.953} C_VEL
LIN {X 0,Y 213.946,Z 156.64,A -85,B 0,C 180,E1 -20682.804,E2 -20682.804} C_VEL
LIN {X 0,Y 213.955,Z 156.639,A -85,B 0,C 180,E1 -20686.707,E2 -20686.707} C_VEL
LIN {X 0,Y 214.144,Z 156.6,A -85,B 0,C 180,E1 -20690.556,E2 -20690.556} C_VEL
LIN {X 0,Y 214.211,Z 156.608,A -85,B 0,C 180,E1 -20692.459,E2 -20692.459} C_VEL
LIN {X 0,Y 214.447,Z 156.561,A -85,B 0,C 180,E1 -20698.122,E2 -20698.122} C_VEL
LIN {X 0,Y 214.549,Z 156.546,A -85,B 0,C 180,E1 -20700,E2 -20700} C_VEL
LIN {X 0,Y 214.448,Z 156.576,A -85,B 0,C 180,E1 -20701.878,E2 -20701.878} C_VEL
LIN {X 0,Y 214.23,Z 156.592,A -85,B 0,C 180,E1 -20707.54,E2 -20707.54} C_VEL
LIN {X 0,Y 214.047,Z 156.624,A -85,B 0,C 180,E1 -20711.362,E2 -20711.362} C_VEL
LIN {X 0,Y 213.937,Z 156.644,A -85,B 0,C 180,E1 -20715.237,E2 -20715.237} C_VEL
LIN {X 0,Y 213.842,Z 156.639,A -85,B 0,C 180,E1 -20719.187,E2 -20719.187} C_VEL
LIN {X 0,Y 213.85,Z 156.658,A -85,B 0,C 180,E1 -20723.227,E2 -20723.227} C_VEL
LIN {X 0,Y 213.831,Z 156.645,A -85,B 0,C 180,E1 -20727.45,E2 -20727.45} C_VEL
LIN {X 0,Y 213.779,Z 156.665,A -85,B 0,C 180,E1 -20731.736,E2 -20731.736} C_VEL
LIN {X 0,Y 213.746,Z 156.671,A -85,B 0,C 180,E1 -20736.288,E2 -20736.288} C_VEL
LIN {X 0,Y 213.714,Z 156.669,A -85,B 0,C 180,E1 -20741.125,E2 -20741.125} C_VEL
LIN {X 0,Y 213.706,Z 156.678,A -85,B 0,C 180,E1 -20743.679,E2 -20743.679} C_VEL
LIN {X 0,Y 213.705,Z 156.643,A -85,B 0,C 180,E1 -20746.345,E2 -20746.345} C_VEL
LIN {X 0,Y 213.738,Z 156.673,A -85,B 0,C 180,E1 -20751.336,E2 -20751.336} C_VEL
LIN {X 0,Y 213.769,Z 156.643,A -85,B 0,C 180,E1 -20756.02,E2 -20756.02} C_VEL
LIN {X 0,Y 213.851,Z 156.868,A -85,B 0,C 180,E1 -20759.004,E2 -20759.004} C_VEL
LIN {X 0,Y 214.222,Z 158.399,A -85,B 0,C 180,E1 -20759.724,E2 -20759.724} C_VEL
LIN {X 0,Y 219.45,Z 169.828,A -85,B 0,C 180,E1 -20761.011,E2 -20761.011} C_VEL
LIN {X 0,Y 224.98,Z 183.582,A -85,B 0,C 180,E1 -20762.281,E2 -20762.281} C_VEL
LIN {X 0,Y 226.5,Z 188.662,A -85,B 0,C 180,E1 -20762.662,E2 -20762.662} C_VEL
LIN {X 0,Y 227.608,Z 196.751,A -85,B 0,C 180,E1 -20763.088,E2 -20763.088} C_VEL
LIN {X 0,Y 226.192,Z 234.974,A -85,B 0,C 180,E1 -20764.298,E2 -20764.298} C_VEL
LIN {X 0,Y 225.43,Z 245.812,A -85,B 0,C 180,E1 -20764.918,E2 -20764.918} C_VEL
LIN {X 0,Y 224.156,Z 257.271,A -85,B 0,C 180,E1 -20765.946,E2 -20765.946} C_VEL
LIN {X 0,Y 222.814,Z 266.078,A -85,B 0,C 180,E1 -20767.024,E2 -20767.024} C_VEL
LIN {X 0,Y 221.375,Z 274.459,A -85,B 0,C 180,E1 -20768.342,E2 -20768.342} C_VEL
LIN {X 0,Y 219.708,Z 282.375,A -85,B 0,C 180,E1 -20769.887,E2 -20769.887} C_VEL
LIN {X 0,Y 218.071,Z 289.755,A -85,B 0,C 180,E1 -20771.686,E2 -20771.686} C_VEL
LIN {X 0,Y 216.255,Z 297.231,A -85,B 0,C 180,E1 -20773.964,E2 -20773.964} C_VEL
LIN {X 0,Y 214.48,Z 304.082,A -85,B 0,C 180,E1 -20776.739,E2 -20776.739} C_VEL
LIN {X 0,Y 213.198,Z 309.259,A -85,B 0,C 180,E1 -20779.554,E2 -20779.554} C_VEL
LIN {X 0,Y 212.514,Z 311.914,A -85,B 0,C 180,E1 -20781.441,E2 -20781.441} C_VEL
LIN {X 0,Y 211.893,Z 314.82,A -85,B 0,C 180,E1 -20784.289,E2 -20784.289} C_VEL
LIN {X 0,Y 211.63,Z 316.088,A -85,B 0,C 180,E1 -20786.191,E2 -20786.191} C_VEL
LIN {X 0,Y 211.476,Z 316.886,A -85,B 0,C 180,E1 -20788.095,E2 -20788.095} C_VEL
LIN {X 0,Y 211.487,Z 317.189,A -85,B 0,C 180,E1 -20790,E2 -20790} C_VEL
LIN {X 0,Y 211.475,Z 316.911,A -85,B 0,C 180,E1 -20791.904,E2 -20791.904} C_VEL
LIN {X 0,Y 211.625,Z 316.161,A -85,B 0,C 180,E1 -20793.808,E2 -20793.808} C_VEL
LIN {X 0,Y 211.862,Z 314.943,A -85,B 0,C 180,E1 -20795.711,E2 -20795.711} C_VEL
LIN {X 0,Y 212.506,Z 312.088,A -85,B 0,C 180,E1 -20798.558,E2 -20798.558} C_VEL
LIN {X 0,Y 213.175,Z 309.487,A -85,B 0,C 180,E1 -20800.446,E2 -20800.446} C_VEL
LIN {X 0,Y 214.455,Z 304.371,A -85,B 0,C 180,E1 -20803.261,E2 -20803.261} C_VEL
LIN {X 0,Y 215.879,Z 298.866,A -85,B 0,C 180,E1 -20805.579,E2 -20805.579} C_VEL
LIN {X 0,Y 217.621,Z 291.945,A -85,B 0,C 180,E1 -20807.866,E2 -20807.866} C_VEL
LIN {X 0,Y 219.413,Z 283.997,A -85,B 0,C 180,E1 -20809.896,E2 -20809.896} C_VEL
LIN {X 0,Y 221.045,Z 276.417,A -85,B 0,C 180,E1 -20811.446,E2 -20811.446} C_VEL
LIN {X 0,Y 222.543,Z 268.469,A -85,B 0,C 180,E1 -20812.759,E2 -20812.759} C_VEL
LIN {X 0,Y 223.878,Z 260.254,A -85,B 0,C 180,E1 -20813.839,E2 -20813.839} C_VEL
LIN {X 0,Y 225.015,Z 251.309,A -85,B 0,C 180,E1 -20814.754,E2 -20814.754} C_VEL
LIN {X 0,Y 225.832,Z 241.813,A -85,B 0,C 180,E1 -20815.476,E2 -20815.476} C_VEL
LIN {X 0,Y 226.456,Z 230.799,A -85,B 0,C 180,E1 -20816.015,E2 -20816.015} C_VEL
LIN {X 0,Y 227.533,Z 194.779,A -85,B 0,C 180,E1 -20817.137,E2 -20817.137} C_VEL
LIN {X 0,Y 226.056,Z 186.515,A -85,B 0,C 180,E1 -20817.62,E2 -20817.62} C_VEL
LIN {X 0,Y 219.989,Z 170.959,A -85,B 0,C 180,E1 -20819.021,E2 -20819.021} C_VEL
LIN {X 0,Y 214.277,Z 158.655,A -85,B 0,C 180,E1 -20820.384,E2 -20820.384} C_VEL
LIN {X 0,Y 213.873,Z 157.149,A -85,B 0,C 180,E1 -20820.984,E2 -20820.984} C_VEL
LIN {X 0,Y 213.78,Z 156.665,A -85,B 0,C 180,E1 -20821.735,E2 -20821.735} C_VEL
LIN {X 0,Y 213.753,Z 156.648,A -85,B 0,C 180,E1 -20826.286,E2 -20826.286} C_VEL
LIN {X 0,Y 213.713,Z 156.642,A -85,B 0,C 180,E1 -20831.124,E2 -20831.124} C_VEL
LIN {X 0,Y 213.703,Z 156.64,A -85,B 0,C 180,E1 -20833.679,E2 -20833.679} C_VEL
LIN {X 0,Y 213.704,Z 156.677,A -85,B 0,C 180,E1 -20836.344,E2 -20836.344} C_VEL
LIN {X 0,Y 213.716,Z 156.667,A -85,B 0,C 180,E1 -20839.142,E2 -20839.142} C_VEL
LIN {X 0,Y 213.743,Z 156.672,A -85,B 0,C 180,E1 -20843.711,E2 -20843.711} C_VEL
LIN {X 0,Y 213.794,Z 156.663,A -85,B 0,C 180,E1 -20848.724,E2 -20848.724} C_VEL
LIN {X 0,Y 213.825,Z 156.646,A -85,B 0,C 180,E1 -20852.603,E2 -20852.603} C_VEL
LIN {X 0,Y 213.851,Z 156.659,A -85,B 0,C 180,E1 -20856.952,E2 -20856.952} C_VEL
LIN {X 0,Y 213.943,Z 156.626,A -85,B 0,C 180,E1 -20862.803,E2 -20862.803} C_VEL
LIN {X 0,Y 213.98,Z 156.643,A -85,B 0,C 180,E1 -20866.708,E2 -20866.708} C_VEL
LIN {X 0,Y 214.166,Z 156.594,A -85,B 0,C 180,E1 -20870.556,E2 -20870.556} C_VEL
LIN {X 0,Y 214.227,Z 156.592,A -85,B 0,C 180,E1 -20872.459,E2 -20872.459} C_VEL
LIN {X 0,Y 214.445,Z 156.576,A -85,B 0,C 180,E1 -20878.122,E2 -20878.122} C_VEL
LIN {X 0,Y 214.549,Z 156.547,A -85,B 0,C 180,E1 -20880,E2 -20880} C_VEL
LIN {X 0,Y 214.445,Z 156.561,A -85,B 0,C 180,E1 -20881.878,E2 -20881.878} C_VEL
LIN {X 0,Y 214.24,Z 156.604,A -85,B 0,C 180,E1 -20887.54,E2 -20887.54} C_VEL
LIN {X 0,Y 214.044,Z 156.611,A -85,B 0,C 180,E1 -20891.362,E2 -20891.362} C_VEL
LIN {X 0,Y 213.933,Z 156.65,A -85,B 0,C 180,E1 -20895.237,E2 -20895.237} C_VEL
LIN {X 0,Y 213.838,Z 156.639,A -85,B 0,C 180,E1 -20899.187,E2 -20899.187} C_VEL
LIN {X 0,Y 213.846,Z 156.66,A -85,B 0,C 180,E1 -20903.227,E2 -20903.227} C_VEL
LIN {X 0,Y 213.828,Z 156.643,A -85,B 0,C 180,E1 -20907.45,E2 -20907.45} C_VEL
LIN {X 0,Y 213.776,Z 156.668,A -85,B 0,C 180,E1 -20911.736,E2 -20911.736} C_VEL
LIN {X 0,Y 213.742,Z 156.666,A -85,B 0,C 180,E1 -20916.288,E2 -20916.288} C_VEL
LIN {X 0,Y 213.709,Z 156.647,A -85,B 0,C 180,E1 -20921.126,E2 -20921.126} C_VEL
LIN {X 0,Y 213.701,Z 156.628,A -85,B 0,C 180,E1 -20923.68,E2 -20923.68} C_VEL
LIN {X 0,Y 213.701,Z 156.664,A -85,B 0,C 180,E1 -20926.345,E2 -20926.345} C_VEL
LIN {X 0,Y 213.715,Z 156.671,A -85,B 0,C 180,E1 -20929.144,E2 -20929.144} C_VEL
LIN {X 0,Y 213.743,Z 156.66,A -85,B 0,C 180,E1 -20933.712,E2 -20933.712} C_VEL
LIN {X 0,Y 213.732,Z 156.671,A -85,B 0,C 180,E1 -20934.288,E2 -20934.288} C_VEL
LIN {X 0,Y 213.591,Z 157.263,A -85,B 0,C 180,E1 -20935.287,E2 -20935.287} C_VEL
LIN {X 0,Y 213.076,Z 159.768,A -85,B 0,C 180,E1 -20936.662,E2 -20936.662} C_VEL
LIN {X 0,Y 212.546,Z 163.533,A -85,B 0,C 180,E1 -20937.846,E2 -20937.846} C_VEL
LIN {X 0,Y 212.31,Z 168.234,A -85,B 0,C 180,E1 -20938.86,E2 -20938.86} C_VEL
LIN {X 0,Y 212.773,Z 173.419,A -85,B 0,C 180,E1 -20939.662,E2 -20939.662} C_VEL
LIN {X 0,Y 213.712,Z 177.001,A -85,B 0,C 180,E1 -20940.057,E2 -20940.057} C_VEL
LIN {X 0,Y 217.49,Z 186.644,A -85,B 0,C 180,E1 -20940.983,E2 -20940.983} C_VEL
LIN {X 0,Y 220.789,Z 209.799,A -85,B 0,C 180,E1 -20942.29,E2 -20942.29} C_VEL
LIN {X 0,Y 219.741,Z 241.272,A -85,B 0,C 180,E1 -20943.334,E2 -20943.334} C_VEL
LIN {X 0,Y 218.993,Z 250.901,A -85,B 0,C 180,E1 -20943.856,E2 -20943.856} C_VEL
LIN {X 0,Y 217.847,Z 260.807,A -85,B 0,C 180,E1 -20944.657,E2 -20944.657} C_VEL
LIN {X 0,Y 216.047,Z 272.482,A -85,B 0,C 180,E1 -20946.008,E2 -20946.008} C_VEL
LIN {X 0,Y 214.412,Z 281.04,A -85,B 0,C 180,E1 -20947.348,E2 -20947.348} C_VEL
LIN {X 0,Y 212.669,Z 289.095,A -85,B 0,C 180,E1 -20948.938,E2 -20948.938} C_VEL
LIN {X 0,Y 211.055,Z 295.749,A -85,B 0,C 180,E1 -20950.55,E2 -20950.55} C_VEL
LIN {X 0,Y 209.438,Z 302.067,A -85,B 0,C 180,E1 -20952.422,E2 -20952.422} C_VEL
LIN {X 0,Y 208.078,Z 307.318,A -85,B 0,C 180,E1 -20954.324,E2 -20954.324} C_VEL
LIN {X 0,Y 206.955,Z 311.697,A -85,B 0,C 180,E1 -20956.249,E2 -20956.249} C_VEL
LIN {X 0,Y 205.685,Z 316.865,A -85,B 0,C 180,E1 -20959.169,E2 -20959.169} C_VEL
LIN {X 0,Y 204.831,Z 320.658,A -85,B 0,C 180,E1 -20962.112,E2 -20962.112} C_VEL
LIN {X 0,Y 204.506,Z 322.4,A -85,B 0,C 180,E1 -20964.083,E2 -20964.083} C_VEL
LIN {X 0,Y 204.342,Z 323.647,A -85,B 0,C 180,E1 -20966.056,E2 -20966.056} C_VEL
LIN {X 0,Y 204.303,Z 324.421,A -85,B 0,C 180,E1 -20968.029,E2 -20968.029} C_VEL
LIN {X 0,Y 204.346,Z 324.714,A -85,B 0,C 180,E1 -20970,E2 -20970} C_VEL
LIN {X 0,Y 204.303,Z 324.412,A -85,B 0,C 180,E1 -20971.972,E2 -20971.972} C_VEL
LIN {X 0,Y 204.354,Z 323.504,A -85,B 0,C 180,E1 -20974.179,E2 -20974.179} C_VEL
LIN {X 0,Y 204.508,Z 322.353,A -85,B 0,C 180,E1 -20975.918,E2 -20975.918} C_VEL
LIN {X 0,Y 205.029,Z 319.435,A -85,B 0,C 180,E1 -20978.874,E2 -20978.874} C_VEL
LIN {X 0,Y 205.631,Z 316.776,A -85,B 0,C 180,E1 -20980.835,E2 -20980.835} C_VEL
LIN {X 0,Y 206.952,Z 311.584,A -85,B 0,C 180,E1 -20983.752,E2 -20983.752} C_VEL
LIN {X 0,Y 208.722,Z 304.737,A -85,B 0,C 180,E1 -20986.632,E2 -20986.632} C_VEL
LIN {X 0,Y 210.65,Z 297.259,A -85,B 0,C 180,E1 -20988.984,E2 -20988.984} C_VEL
LIN {X 0,Y 212.443,Z 289.885,A -85,B 0,C 180,E1 -20990.832,E2 -20990.832} C_VEL
LIN {X 0,Y 214.153,Z 281.985,A -85,B 0,C 180,E1 -20992.427,E2 -20992.427} C_VEL
LIN {X 0,Y 215.783,Z 273.633,A -85,B 0,C 180,E1 -20993.769,E2 -20993.769} C_VEL
LIN {X 0,Y 217.497,Z 262.73,A -85,B 0,C 180,E1 -20995.12,E2 -20995.12} C_VEL
LIN {X 0,Y 218.885,Z 251.263,A -85,B 0,C 180,E1 -20996.071,E2 -20996.071} C_VEL
LIN {X 0,Y 219.696,Z 241.394,A -85,B 0,C 180,E1 -20996.607,E2 -20996.607} C_VEL
LIN {X 0,Y 220.703,Z 209.638,A -85,B 0,C 180,E1 -20997.667,E2 -20997.667} C_VEL
LIN {X 0,Y 217.241,Z 185.966,A -85,B 0,C 180,E1 -20999.015,E2 -20999.015} C_VEL
LIN {X 0,Y 211.274,Z 171.379,A -85,B 0,C 180,E1 -21000.473,E2 -21000.473} C_VEL
LIN {X 0,Y 208.341,Z 164.809,A -85,B 0,C 180,E1 -21001.264,E2 -21001.264} C_VEL
LIN {X 0,Y 207.21,Z 159.765,A -85,B 0,C 180,E1 -21004.031,E2 -21004.031} C_VEL
LIN {X 0,Y 206.705,Z 157.567,A -85,B 0,C 180,E1 -21005.512,E2 -21005.512} C_VEL
LIN {X 0,Y 206.661,Z 157.542,A -85,B 0,C 180,E1 -21010.252,E2 -21010.252} C_VEL
LIN {X 0,Y 206.631,Z 157.523,A -85,B 0,C 180,E1 -21014.418,E2 -21014.418} C_VEL
LIN {X 0,Y 206.641,Z 157.519,A -85,B 0,C 180,E1 -21018.438,E2 -21018.438} C_VEL
LIN {X 0,Y 206.681,Z 157.553,A -85,B 0,C 180,E1 -21022.261,E2 -21022.261} C_VEL
LIN {X 0,Y 206.704,Z 157.544,A -85,B 0,C 180,E1 -21027.043,E2 -21027.043} C_VEL
LIN {X 0,Y 206.768,Z 157.52,A -85,B 0,C 180,E1 -21032.097,E2 -21032.097} C_VEL
LIN {X 0,Y 206.787,Z 157.54,A -85,B 0,C 180,E1 -21036.584,E2 -21036.584} C_VEL
LIN {X 0,Y 206.875,Z 157.516,A -85,B 0,C 180,E1 -21042.197,E2 -21042.197} C_VEL
LIN {X 0,Y 206.898,Z 157.522,A -85,B 0,C 180,E1 -21046.245,E2 -21046.245} C_VEL
LIN {X 0,Y 207.101,Z 157.473,A -85,B 0,C 180,E1 -21050.231,E2 -21050.231} C_VEL
LIN {X 0,Y 207.068,Z 157.505,A -85,B 0,C 180,E1 -21054.156,E2 -21054.156} C_VEL
LIN {X 0,Y 207.384,Z 157.44,A -85,B 0,C 180,E1 -21058.058,E2 -21058.058} C_VEL
LIN {X 0,Y 207.514,Z 157.421,A -85,B 0,C 180,E1 -21060,E2 -21060} C_VEL
LIN {X 0,Y 207.384,Z 157.455,A -85,B 0,C 180,E1 -21061.942,E2 -21061.942} C_VEL
LIN {X 0,Y 207.171,Z 157.468,A -85,B 0,C 180,E1 -21067.799,E2 -21067.799} C_VEL
LIN {X 0,Y 206.984,Z 157.506,A -85,B 0,C 180,E1 -21071.755,E2 -21071.755} C_VEL
LIN {X 0,Y 206.87,Z 157.52,A -85,B 0,C 180,E1 -21075.771,E2 -21075.771} C_VEL
LIN {X 0,Y 206.786,Z 157.523,A -85,B 0,C 180,E1 -21079.869,E2 -21079.869} C_VEL
LIN {X 0,Y 206.766,Z 157.537,A -85,B 0,C 180,E1 -21084.072,E2 -21084.072} C_VEL
LIN {X 0,Y 206.747,Z 157.536,A -85,B 0,C 180,E1 -21088.419,E2 -21088.419} C_VEL
LIN {X 0,Y 206.704,Z 157.534,A -85,B 0,C 180,E1 -21092.957,E2 -21092.957} C_VEL
LIN {X 0,Y 206.682,Z 157.552,A -85,B 0,C 180,E1 -21097.74,E2 -21097.74} C_VEL
LIN {X 0,Y 206.644,Z 157.553,A -85,B 0,C 180,E1 -21101.563,E2 -21101.563} C_VEL
LIN {X 0,Y 206.633,Z 157.532,A -85,B 0,C 180,E1 -21105.582,E2 -21105.582} C_VEL
LIN {X 0,Y 206.667,Z 157.529,A -85,B 0,C 180,E1 -21109.75,E2 -21109.75} C_VEL
LIN {X 0,Y 206.734,Z 157.516,A -85,B 0,C 180,E1 -21114.695,E2 -21114.695} C_VEL
LIN {X 0,Y 206.773,Z 157.719,A -85,B 0,C 180,E1 -21118.182,E2 -21118.182} C_VEL
